	// always
	SIf.Cur.dinPosition_0_1deg := LREAL_TO_DINT(In_pAD_SIf^.stMove.lreActPos)*10;
	SIf.Cur.dinModPosition_0_1deg := LREAL_TO_DINT(In_pAD_SIf^.stMove.lreActModPos)*10;
	SIf.Cur.dinSpeed_0_1deg_s := LREAL_TO_DINT(In_pAD_SIf^.stMove.lreActVel)*10;
	SIf.Cur.dinTorque_0_1Nm := LREAL_TO_DINT(In_pAD_SIf^.stMove.lreActTorque)*10;
	SIf.Cur.bol_di1 := In_pAD_SIf^.stStatus.stDigIn.bol_SI0;
	SIf.Cur.bol_di2 := In_pAD_SIf^.stStatus.stDigIn.bol_SI1;
	SIf.Cur.bol_di3 := In_pAD_SIf^.stStatus.stDigIn.bol_SI2;
	SIf.Cur.bol_di4 := In_pAD_SIf^.stStatus.stDigIn.bol_SI3; // used for homing.....

	// info message 'software limit reached'
	IF ((In_pAD_SIf^.stStatus.bolNegSWSwitch) OR (In_pAD_SIf^.stStatus.bolPosSWSwitch)) THEN 
		IF (SIf.Alm[E_ALM_RAX.SwLimit].bol=FALSE)THEN
			// 'software limit reached';
			pfbAlarmCtrl^.setAlarm(CIf.Info.intCtrlId,E_ALM_RAX.SwLimit,0,ADR(SIf.Alm),E_AlmState.SET,CIf.Job.eMe_ActivAlmClass);
			SIf.Alm[E_ALM_RAX.SwLimit].bol:= TRUE;
		END_IF;
	ELSE
		IF (SIf.Alm[E_ALM_RAX.SwLimit].bol) THEN
			pfbAlarmCtrl^.setAlarm(CIf.Info.intCtrlId,4,0,ADR(SIf.Alm),E_AlmState.CLR,CIf.Job.eMe_ActivAlmClass);
			SIf.Alm[E_ALM_RAX.SwLimit].bol:= FALSE;
		END_IF
	END_IF
	
	//------------------------------------------------------------------------------------------------------------------------------------
	// set parameter
	// in Manual set % speed to 100% for single cmd's
	IF (CIf.Job.eMode=E_Mode.MANU) THEN
		SIf.Par.dinSpeed_per := 100;
		SIf.Par.dinAcc_per := 100;
		SIf.Par.dinDec_per := 100;
	END_IF	
	
	In_pAD_SIf^.stMove.lreSetSpeed := fSetPar(SIf.Par.dinSpeed_0_1deg_s,SIf.Par.dinSpeed_per);
	In_pAD_SIf^.stMove.lreSetAcc := fSetPar(SIf.Par.dintAccDec_0_1deg_s2,SIf.Par.dinAcc_per);
	In_pAD_SIf^.stMove.lreSetDec := fSetPar(SIf.Par.dintAccDec_0_1deg_s2,SIf.Par.dinDec_per);
	IF (SIf.Par.dinSetDecFast_0_1deg_s2>0) THEN
		In_pAD_SIf^.stMove.lreSetDecFast := DINT_TO_LREAL(SIf.Par.dinSetDecFast_0_1deg_s2)/10.0;
	ELSE
		In_pAD_SIf^.stMove.lreSetDecFast := In_pAD_SIf^.stMove.lreSetDec;
	END_IF
	In_pAD_SIf^.stCfg.bolSimulation := CIf.SwCfg.bolSimulation;
	
	// ----------------------------------------------------------------------------------
	// Conditions Always
	IF (me.StateMachine.intState>cSTA_PON) THEN	
		IF ((In_pAD_SIf^.stErr.bolErrorActive) AND (me.StateMachine.intState<>cSTA_ERROR) AND (me.StateMachine.intState<>cSTA_ERRORQuit)) THEN
			// detect drive error
			me.StateMachine.intStateNext := cSTA_ERROR;
		END_IF
	END_IF
END_IF
END_METHOD

PROPERTY PUBLIC CtrlSIf : POINTER TO T_Ctrl_SIf_RAX
GET
CtrlSIf := ADR(SIf);
END_GET
END_PROPERTY

{attribute 'object_name' := 'FB_init'}
METHOD FB_init : BOOL
VAR_INPUT
	///if TRUE, the retain variables are initialized (warm start / cold start)
	bInitRetains: BOOL;
	///if TRUE, the instance afterwards gets moved into the copy code (online change)
	bInCopyCode: BOOL;
END_VAR
VAR
	udiTaskCnt: UDINT;
END_VAR
//------------------------------------------------------------------------------------------------------------------------
// to manually change in new FUB implementation!!!
// define valid commands for this controller
FOR ii:= 0 TO (SIZEOF(CIf.Job.aCmdList)/SIZEOF(CIf.Job.aCmdList[0])-1) BY 1 DO
	IF (CIf.Job.aCmdList[ii].intCmd=cCMD_INITIALIZED) THEN
		// found first empty array element
		EXIT;
	END_IF
END_FOR
CIf.Job.aCmdList[ii].intCmd := cCMD_INIT;
CIf.Job.aCmdList[ii].strName := 'Init'; 
CIf.Job.aCmdList[ii].bolAvailable := TRUE;
ii := ii +1;
CIf.Job.aCmdList[ii].intCmd := RAX_CmdState.cCMD_POS;
CIf.Job.aCmdList[ii].strName := 'Position absolute';
CIf.Job.aCmdList[ii].bolAvailable := TRUE;
ii := ii +1;
CIf.Job.aCmdList[ii].intCmd := RAX_CmdState.cCMD_JOG_NEG;
CIf.Job.aCmdList[ii].strName := 'jogging negativ direction';
CIf.Job.aCmdList[ii].bolAvailable := TRUE;
ii := ii +1;
CIf.Job.aCmdList[ii].intCmd := RAX_CmdState.cCMD_JOG_POS;
CIf.Job.aCmdList[ii].strName := 'jogging positive direction';
CIf.Job.aCmdList[ii].bolAvailable := TRUE;
ii := ii +1;
CIf.Job.aCmdList[ii].intCmd := RAX_CmdState.cCMD_HOME;
CIf.Job.aCmdList[ii].strName := 'Home';
CIf.Job.aCmdList[ii].bolAvailable := TRUE;
ii := ii +1;
CIf.Job.aCmdList[ii].intCmd := RAX_CmdState.cCMD_REL_POS;
CIf.Job.aCmdList[ii].strName := 'Relative move';
CIf.Job.aCmdList[ii].bolAvailable := TRUE;
ii := ii +1;
CIf.Job.aCmdList[ii].intCmd := RAX_CmdState.cCMD_TURN;
CIf.Job.aCmdList[ii].strName := 'Turn';
CIf.Job.aCmdList[ii].bolAvailable := TRUE;
ii := ii +1;

// set name of class/typ
CIf.Info.strType := 'FB_RAX';
CIf.Info.strFullName := 'Rotative Axis';

// set alarm class
SIf.Alm[E_ALM_RAX.GeneralDrive].eAlmClass := E_AlmClass.OFF;
SIf.Alm[E_ALM_RAX.GeneralDrive].strText := 'general drive failure -> info number'; 
SIf.Alm[E_ALM_RAX.GeneralNc].eAlmClass := E_AlmClass.OFF;
SIf.Alm[E_ALM_RAX.GeneralNc].strText := 'general nc failure -> info number';
SIf.Alm[E_ALM_RAX.SwLimit].eAlmClass := E_AlmClass.INFO;
SIf.Alm[E_ALM_RAX.SwLimit].strText := 'software limit reached';
SIf.Alm[E_ALM_RAX.NegHwLimit].eAlmClass := E_AlmClass.OFF;
SIf.Alm[E_ALM_RAX.NegHwLimit].strText := 'neg. hardware switch detected';
SIf.Alm[E_ALM_RAX.PosHwLimit].eAlmClass := E_AlmClass.OFF;
SIf.Alm[E_ALM_RAX.PosHwLimit].strText := 'pos. hardware switch detected';
SIf.Alm[E_ALM_RAX.InterlockNegMove].eAlmClass := E_AlmClass.EOFF;
SIf.Alm[E_ALM_RAX.InterlockNegMove].strText := 'interlock neg. movement - movement stopped';
SIf.Alm[E_ALM_RAX.InterlockPosMove].eAlmClass := E_AlmClass.EOFF;
SIf.Alm[E_ALM_RAX.InterlockPosMove].strText := 'interlock pos. movement  - movement stopped';
SIf.Alm[E_ALM_RAX.GeneralMCFUB].eAlmClass := E_AlmClass.STOP;
SIf.Alm[E_ALM_RAX.GeneralMCFUB].strText := 'MC fub error -> info number';

//*******************************************************************************
// initial values
//*******************************************************************************

// software configuration
CIf.SwCfg.bolExist := TRUE;
CIf.SwCfg.bolSimulation := FALSE;

// cfg
//SIf.Cfg.eHomingMode := MC_HomingMode.MC_Direct;
SIf.Cfg.eHomingMode := MC_HomingMode.MC_DefaultHoming;
SIf.Cfg.lreShortestWayWindow_deg := 20.0; //20.0°

// parmeter
SIf.Par.dinHomeOffset_0_1deg := -900;
SIf.Par.dinPos_0_1deg := 0;
SIf.Par.dinRelDist_0_1deg := 10;
SIf.Par.dinPositionInit_0_1deg := 0;
SIf.Par.dintAccDec_0_1deg_s2 := 4000;
SIf.Par.dinAcc_per := 100;
SIf.Par.dinDec_per := 100;
SIf.Par.dinSetDecFast_0_1deg_s2 := 4000;
SIf.Par.dinSpeed_0_1deg_s := 200;
SIf.Par.dinSpeed_per := 200;
SIf.Par.dinSWLimitNeg_0_1deg := 0;
SIf.Par.dinSWLimitPos_0_1deg := 360;
END_METHOD

{attribute 'object_name' := 'getCmdState'}
METHOD PROTECTED getCmdState : STRING
VAR_INPUT
	intCmdState: INT;
	bolState: BOOL;
END_VAR
getCmdState := SUPER^.getCmdState(intCmdState:=intCmdState,bolState:=bolState); // get global/base defined cmds/states
IF (getCmdState='') THEN // global not defined get local
	// get string cmd/state string information in runtime
	IF (bolState=FALSE) THEN
		// cmd's
		CASE intCmdState OF
			RAX_CmdState.cCMD_HOME: 
				getCmdState := 'cCMD_HOME';
			RAX_CmdState.cCMD_POS: 
				getCmdState := 'cCMD_POS';
			RAX_CmdState.cCMD_JOG_NEG: 
				getCmdState := 'cCMD_JOG_NEG';
			RAX_CmdState.cCMD_JOG_POS: 
				getCmdState := 'cCMD_JOG_POS';
			RAX_CmdState.cCMD_REL_POS: 
				getCmdState := 'cCMD_REL_POS';
			RAX_CmdState.cCMD_TURN: 
				getCmdState := 'cCMD_TURN';
		ELSE
				getCmdState := 'not defined';
		END_CASE;
	ELSE
	
	// cmd's
		CASE intCmdState OF
			RAX_CmdState.cSTA_POSBusy: 
				getCmdState := 'cSTA_POSBusy';
			RAX_CmdState.cSTA_POS: 
				getCmdState := 'cSTA_POS';
			RAX_CmdState.cSTA_JOG_NEG: 
				getCmdState := 'cSTA_JOG_NEG';
			RAX_CmdState.cSTA_JOG_POS: 
				getCmdState := 'cSTA_JOG_POS';
			RAX_CmdState.cSTA_REL_POSBusy: 
				getCmdState := 'cSTA_REL_POSBusy';
			RAX_CmdState.cSTA_REL_POS: 
				getCmdState := 'cSTA_REL_POS';
			RAX_CmdState.cSTA_TURNBusy: 
				getCmdState := 'cSTA_TURNBusy';
			RAX_CmdState.cSTA_TURN: 
				getCmdState := 'cSTA_TURN';			
			cSUB_WriteSW: 
				getCmdState := 'cSUB_WriteSW';
			cSUB_Home: 
				getCmdState := 'cSUB_Home';
			cSUB_MoveToInitPos: 
				getCmdState := 'cSUB_MoveToInitPos';
			cSUB_Finished: 
				getCmdState := 'cSUB_Finished';
			cSUB_INITIALIZED:
				getCmdState := 'cSUB_INITIALIZED';
		ELSE
				getCmdState := 'not defined';
		END_CASE;
	END_IF
END_IF
END_METHOD

{attribute 'object_name' := 'getDirection'}
METHOD PROTECTED getDirection : MC_Direction
VAR_INPUT
	dinActualPosition: DINT;
	lreSetPosition: LREAL;
END_VAR
VAR
	Direction: MC_Direction;
	lreActualPosition: LREAL;
END_VAR
Direction := MC_Positive_Direction;	// MC_Shortest_Way, MC_Negative_Direction, 
lreActualPosition := DINT_TO_LREAL(dinActualPosition)/10.0;
IF (ABS(ABS(lreActualPosition) - ABS(lreSetPosition)) <= SIf.Cfg.lreShortestWayWindow_deg) THEN
	Direction := MC_Shortest_Way;
ELSIF (lreActualPosition < 0) THEN
	Direction := MC_Negative_Direction;
END_IF;

getDirection := Direction;
END_METHOD

{attribute 'object_name' := 'IoOutBridge'}
METHOD PROTECTED IoOutBridge : BOOL
// digitale and analoge inputs read from hardware or forcing
IF (CIf.SwCfg.bolSimulation = FALSE) THEN
	// check interlocks to prevent damages
	IF (CIf.Job.bolIlkOverwrite=FALSE) THEN
		IF (SIf.Ilk.bolMovePos) AND (In_pAD_SIf^.stStatus.bolCtrlOn)  AND ((In_pAD_SIf^.intCmd=cPOD_CMD_POS_JOG) OR (In_pAD_SIf^.intCmd=cPOD_CMD_POS_MOVE) OR
			((In_pAD_SIf^.stMove.lreSetPos > In_pAD_SIf^.stMove.lreActPos) AND (In_pAD_SIf^.intCmd=cPOD_CMD_ABS_MOVE)) OR
			((In_pAD_SIf^.intCmd=cPOD_CMD_REL_MOVE) AND (In_pAD_SIf^.stMove.lreSetPos>0)) OR (SIf.Cur.dinSpeed_0_1deg_s>5)  )THEN	
			// SIf.Alm[8].strText := 'interlock pos. movement  - movement stopped';
			pfbAlarmCtrl^.setAlarm(CIf.Info.intCtrlId,E_ALM_RAX.InterlockPosMove,0,ADR(SIf.Alm),E_AlmState.RST,CIf.Job.eMe_ActivAlmClass);
			In_pAD_SIf^.intCmd:=cPOD_CMD_EMCY_STOP_CTRL_OFF;
		END_IF
		IF (SIf.Ilk.bolMoveNeg) AND (In_pAD_SIf^.stStatus.bolCtrlOn)  AND ((In_pAD_SIf^.intCmd=cPOD_CMD_NEG_JOG) OR (In_pAD_SIf^.intCmd=cPOD_CMD_NEG_MOVE) OR
		 	(In_pAD_SIf^.intCmd=cPOD_CMD_HOME) OR
			((In_pAD_SIf^.stMove.lreSetPos < In_pAD_SIf^.stMove.lreActPos) AND (In_pAD_SIf^.intCmd=cPOD_CMD_ABS_MOVE)) OR
			((In_pAD_SIf^.intCmd=cPOD_CMD_REL_MOVE) AND (In_pAD_SIf^.stMove.lreSetPos<0)) OR (SIf.Cur.dinSpeed_0_1deg_s<-5)  )THEN		
			// 'interlock neg. movement - movement stopped';
			pfbAlarmCtrl^.setAlarm(CIf.Info.intCtrlId,E_ALM_RAX.InterlockNegMove,0,ADR(SIf.Alm),E_AlmState.RST,CIf.Job.eMe_ActivAlmClass);
			In_pAD_SIf^.intCmd:=cPOD_CMD_EMCY_STOP_CTRL_OFF;
		END_IF	
	END_IF

END_IF
END_METHOD

{attribute 'object_name' := 'sta_EOFF'}
METHOD PROTECTED sta_EOFF : BOOL
// state implemetation
//--------------------------------------------------------------------------------------
// Entry action
	IF (me.StateMachine.intState<>me.StateMachine.intStateLastCycle) THEN
		me.StateMachine.intStateLastCycle := me.StateMachine.intState;
		
	END_IF


//--------------------------------------------------------------------------------------
// Cyclic action
	IF (me.StateMachine.intState=me.StateMachine.intStateLastCycle) THEN
		
		// State Change Condition
		IF (me.intCmd<>cCMD_EOFF) AND (me.intCmd<>cCMD_DONE)  AND (me.Alarm.eActivAlmClass<>E_AlmClass.EOFF) THEN
			me.StateMachine.intStateNext := cSTA_OFFBusy;
		END_IF
	END_IF




//--------------------------------------------------------------------------------------
// Exit action
	IF (me.StateMachine.intState<>me.StateMachine.intStateNext) THEN
		;
	END_IF
END_METHOD

{attribute 'object_name' := 'sta_EOFFBusy'}
METHOD PROTECTED sta_EOFFBusy : BOOL
// state implemetation
//--------------------------------------------------------------------------------------
// Entry action
	IF (me.StateMachine.intState<>me.StateMachine.intStateLastCycle) THEN
		me.StateMachine.intStateLastCycle := me.StateMachine.intState;
				
		In_pAD_SIf^.intCmd := cPOD_CMD_EMCY_STOP_CTRL_OFF;
		
	END_IF


//--------------------------------------------------------------------------------------
// Cyclic action
	IF (me.StateMachine.intState=me.StateMachine.intStateLastCycle) THEN
		
		// Simulation
		IF (CIf.SwCfg.bolSimulation) THEN
			;
		END_IF
	
		// no change action
	
		// State Change Condition
		IF (In_pAD_SIf^.intCmd=cPOD_CMD_DONE) AND (In_pAD_SIf^.stStatus.bolCtrlOn=FALSE) THEN
			me.StateMachine.intStateNext := cSTA_EOFF;
		END_IF
	END_IF




//--------------------------------------------------------------------------------------
// Exit action
	IF (me.StateMachine.intState<>me.StateMachine.intStateNext) THEN
		;
	END_IF
END_METHOD

{attribute 'object_name' := 'sta_ERROR'}
METHOD PROTECTED sta_ERROR : BOOL
// state implemetation
//--------------------------------------------------------------------------------------
// Entry action
	IF (me.StateMachine.intState<>me.StateMachine.intStateLastCycle) THEN
		me.StateMachine.intStateHistory := me.StateMachine.intStateLastCycle; // -> possibillity to go back to state before error
		me.StateMachine.intStateLastCycle := me.StateMachine.intState;
		
		
		IF (In_pAD_SIf^.stErr.bolNCError) THEN
			// := 'general nc failure -> info number';
			pfbAlarmCtrl^.setAlarm(CIf.Info.intCtrlId,E_ALM_RAX.GeneralNc,DWORD_TO_DINT(In_pAD_SIf^.stErr.dwoErrorID),ADR(SIf.Alm),E_AlmState.RST,CIf.Job.eMe_ActivAlmClass);
		ELSIF (In_pAD_SIf^.stErr.bolMCError) THEN // to define
			//'MC fub error -> info number';
			pfbAlarmCtrl^.setAlarm(CIf.Info.intCtrlId,E_ALM_RAX.GeneralMCFUB,DWORD_TO_DINT(In_pAD_SIf^.stErr.dwoErrorID),ADR(SIf.Alm),E_AlmState.RST,CIf.Job.eMe_ActivAlmClass);
		ELSIF(In_pAD_SIf^.stErr.dwoErrorID=32000) THEN // Limit switch during movement
			IF (In_pAD_SIf^.stStatus.bolNegHWSwitch) THEN
				// 'neg. hardware switch detected';
				pfbAlarmCtrl^.setAlarm(CIf.Info.intCtrlId,E_ALM_RAX.NegHwLimit,0,ADR(SIf.Alm),E_AlmState.RST,CIf.Job.eMe_ActivAlmClass);
			ELSE
				// 'pos. hardware switch detected';
				pfbAlarmCtrl^.setAlarm(CIf.Info.intCtrlId,E_ALM_RAX.PosHwLimit,0,ADR(SIf.Alm),E_AlmState.RST,CIf.Job.eMe_ActivAlmClass);
			END_IF
		ELSE
			// 'general drive failure -> info number'; 
			pfbAlarmCtrl^.setAlarm(CIf.Info.intCtrlId,E_ALM_RAX.GeneralDrive,DWORD_TO_DINT(In_pAD_SIf^.stErr.dwoErrorID),ADR(SIf.Alm),E_AlmState.RST,CIf.Job.eMe_ActivAlmClass);
		END_IF
			
	END_IF


//--------------------------------------------------------------------------------------
// Cyclic action
	IF (me.StateMachine.intState=me.StateMachine.intStateLastCycle) THEN

		// State Change Condition
		IF (CIf.Job.bolAlmReset = TRUE) THEN
			me.StateMachine.intStateNext := cSTA_ERRORQuit;
		END_IF
	END_IF




//--------------------------------------------------------------------------------------
// Exit action
	IF (me.StateMachine.intState<>me.StateMachine.intStateNext) THEN
		;
	END_IF
END_METHOD

{attribute 'object_name' := 'sta_ERRORQuit'}
METHOD PROTECTED sta_ERRORQuit : BOOL
// state implemetation
//--------------------------------------------------------------------------------------
// Entry action
	IF (me.StateMachine.intState<>me.StateMachine.intStateLastCycle) THEN
		me.StateMachine.intStateLastCycle := me.StateMachine.intState;
		
	END_IF


//--------------------------------------------------------------------------------------
// Cyclic action
	IF (me.StateMachine.intState=me.StateMachine.intStateLastCycle) THEN
		
		;
		// evtl. wait time if reset of device is necessary and then decide to go to states or ERROR state
		IF (CIf.Job.bolAlmReset = TRUE) THEN
			In_pAD_SIf^.stErr.bolErrAck := TRUE; // reset drive error
			CIf.Job.eMe_ActivAlmClass := E_AlmClass.NONE; // reset feedback channel for parent
			CIf.Job.bolAlmReset := FALSE;
		END_IF
		
		// State Change Condition
		IF (In_pAD_SIf^.stErr.bolErrAck = FALSE) THEN // reset done on drive
			IF (me.StateMachine.intStateHistory<=cSTA_PON) THEN
				me.StateMachine.intStateNext := cSTA_PONBusy;
			ELSE
				me.StateMachine.intStateNext := cSTA_OFFBusy;
			END_IF
		END_IF
	END_IF




//--------------------------------------------------------------------------------------
// Exit action
	IF (me.StateMachine.intState<>me.StateMachine.intStateNext) THEN
		;
	END_IF
END_METHOD

{attribute 'object_name' := 'sta_INIT'}
METHOD PROTECTED sta_INIT : BOOL
// state implemetation
//--------------------------------------------------------------------------------------
// Entry action
	IF (me.StateMachine.intState<>me.StateMachine.intStateLastCycle) THEN
		me.StateMachine.intStateLastCycle := me.StateMachine.intState;
		
	END_IF


//--------------------------------------------------------------------------------------
// Cyclic action
	IF (me.StateMachine.intState=me.StateMachine.intStateLastCycle) THEN
		
		;
		
		// State Change Condition
		// check if no important alarm activ
		IF (me.intCmd=RAX_CmdState.cCMD_POS) THEN 
			me.StateMachine.intStateNext := RAX_CmdState.cSTA_POSBusy;
		ELSIF(me.intCmd=RAX_CmdState.cCMD_REL_POS) THEN
				me.StateMachine.intStateNext := RAX_CmdState.cSTA_REL_POSBusy;
		ELSIF(me.intCmd=RAX_CmdState.cCMD_JOG_NEG) THEN
			me.StateMachine.intStateNext := RAX_CmdState.cSTA_JOG_NEG;
		ELSIF(me.intCmd=RAX_CmdState.cCMD_JOG_POS) THEN
			me.StateMachine.intStateNext := RAX_CmdState.cSTA_JOG_POS;
		ELSIF (me.intCmd=RAX_CmdState.cCMD_TURN) THEN 
			me.StateMachine.intStateNext := RAX_CmdState.cSTA_TURNBusy;
		ELSIF (me.intCmd=cCMD_STOP) THEN 
			me.StateMachine.intStateNext := cSTA_STOPBusy;
		END_IF
	END_IF




//--------------------------------------------------------------------------------------
// Exit action
	IF (me.StateMachine.intState<>me.StateMachine.intStateNext) THEN
		;
	END_IF
END_METHOD

{attribute 'object_name' := 'sta_INITBusy'}
METHOD PROTECTED sta_INITBusy : BOOL
// state implemetation
//--------------------------------------------------------------------------------------
// Entry action
	IF (me.StateMachine.intState<>me.StateMachine.intStateLastCycle) THEN
		me.StateMachine.intStateLastCycle := me.StateMachine.intState;

		me.SubStateMachine.intState := cSUB_INITIALIZED; // reset sub statemachine
		me.SubStateMachine.intStateLastCycle := me.SubStateMachine.intState-1;
		me.SubStateMachine.intStateNext := me.SubStateMachine.intState;	
	END_IF


//--------------------------------------------------------------------------------------
// Cyclic action
	IF (me.StateMachine.intState=me.StateMachine.intStateLastCycle) THEN
		
		// Simulation
		IF (CIf.SwCfg.bolSimulation) THEN
			;
		END_IF
	
		// no change action
		// ---------------------------------------------------------------------------------------------------------------------------
		// sub state machine for sequence
		CASE me.SubStateMachine.intState OF
			//--------------------------------------------------------------------------------------
			cSUB_INITIALIZED:
				// Entry action
				IF (me.SubStateMachine.intState<>me.SubStateMachine.intStateLastCycle) THEN
					me.SubStateMachine.intStateLastCycle := me.SubStateMachine.intState;
				END_IF	
				
				// -------------------------------- State Change Condition
				IF(TRUE) THEN
					me.SubStateMachine.intStateNext := cSUB_WriteSW;
				END_IF
					
			//--------------------------------------------------------------------------------------
			cSUB_WriteSW:
				// Entry action
				IF (me.SubStateMachine.intState<>me.SubStateMachine.intStateLastCycle) THEN
					me.SubStateMachine.intStateLastCycle := me.SubStateMachine.intState;
				END_IF	
				
				(*
				// write sw offset to nc system offset to real axis system/encoder!!!!!!!!
				IF ((SIf.Par.lreHomeOffset_mm<>In_pAD_SIf^.stcfg.lreHomePosition) AND (In_pAD_SIf^.intServiceCmd=cPOD_CMD_DONE)) THEN
					In_pAD_SIf^.stService.eNC_ParNumber := MC_AxisParameter.AxisEncoderOffset;
					In_pAD_SIf^.stService.strValue := LREAL_TO_STRING(SIf.Par.lreHomeOffset_mm);
					In_pAD_SIf^.intServiceCmd := cPOD_SCMD_WRITE_PARA_NC;
					In_pAD_SIf^.stcfg.lreHomePosition := SIf.Par.lreHomeOffset_mm;
				END_IF
				
				// write sw-limits to nc system
				IF ((SIf.Par.lreSWLimitNeg_mm<>In_pAD_SIf^.stMove.lreSWLimitNeg_mm) AND (In_pAD_SIf^.intServiceCmd=cPOD_CMD_DONE)) THEN
					In_pAD_SIf^.stService.eNC_ParNumber := MC_AxisParameter.SWLimitNeg;
					In_pAD_SIf^.stService.strValue := LREAL_TO_STRING(SIf.Par.lreSWLimitNeg_mm);
					In_pAD_SIf^.intServiceCmd := cPOD_SCMD_WRITE_PARA_NC;
					In_pAD_SIf^.stMove.lreSWLimitNeg_mm := SIf.Par.lreSWLimitNeg_mm;
				END_IF
				
				IF ((SIf.Par.lreSWLimitPos_mm<>In_pAD_SIf^.stMove.lreSWLimitPos_mm) AND (In_pAD_SIf^.intServiceCmd=cPOD_CMD_DONE)) THEN
					In_pAD_SIf^.stService.eNC_ParNumber := MC_AxisParameter.SWLimitPos;
					In_pAD_SIf^.stService.strValue := LREAL_TO_STRING(SIf.Par.lreSWLimitPos_mm);
					In_pAD_SIf^.intServiceCmd := cPOD_SCMD_WRITE_PARA_NC;
					In_pAD_SIf^.stMove.lreSWLimitPos_mm := SIf.Par.lreSWLimitPos_mm;
				END_IF
*)
				// -------------------------------- State Change Condition
				IF (In_pAD_SIf^.intServiceCmd=cPOD_CMD_DONE) THEN
					IF ((me.intCmd=RAX_CmdState.cCMD_HOME) OR (In_pAD_SIf^.stStatus.bolHomeOk=FALSE)) THEN
						me.SubStateMachine.intStateNext := cSUB_Home;
					ELSIF (me.intCmd=cCMD_INIT) THEN
						me.SubStateMachine.intStateNext := cSUB_MoveToInitPos;
					ELSE
						me.SubStateMachine.intStateNext := cSUB_Finished; // no movement to init position no cmd INIT or HOME
					END_IF;
				END_IF
					
			//--------------------------------------------------------------------------------------
			cSUB_Home:
				// Entry action
				IF (me.SubStateMachine.intState<>me.SubStateMachine.intStateLastCycle) THEN
					me.SubStateMachine.intStateLastCycle := me.SubStateMachine.intState;
		
					In_pAD_SIf^.stCfg.eHomingMode := SIf.Cfg.eHomingMode;
					In_pAD_SIf^.stCfg.lreHomePosition := DINT_TO_LREAL(SIf.Par.dinHomeOffset_0_1deg)/10.0;
					In_pAD_SIf^.intCmd := cPOD_CMD_HOME;	// start homing
	
				END_IF
					
				// State Change Condition
				IF (In_pAD_SIf^.stStatus.bolHomeOk) AND (In_pAD_SIf^.intCmd=cPOD_CMD_DONE) THEN
					me.SubStateMachine.intStateNext := cSUB_MoveToInitPos;
				END_IF
				
			//--------------------------------------------------------------------------------------
			cSUB_MoveToInitPos:
				// Entry action
				IF (me.SubStateMachine.intState<>me.SubStateMachine.intStateLastCycle) THEN
					me.SubStateMachine.intStateLastCycle := me.SubStateMachine.intState;
				
					In_pAD_SIf^.stMove.lreSetPos := DINT_TO_LREAL(SIf.Par.dinPositionInit_0_1deg)/10.0;
					In_pAD_SIf^.stMove.eDirection := getDirection(dinActualPosition:=SIf.Cur.dinModPosition_0_1deg,lreSetPosition:=In_pAD_SIf^.stMove.lreSetPos);
					//In_pAD_SIf^.intCmd := cPOD_CMD_MOD_MOVE;	// absolute position
					In_pAD_SIf^.intCmd := cPOD_CMD_ABS_MOVE;	// absolute position
				END_IF
						
				// State Change Condition
				IF (In_pAD_SIf^.stStatus.bolInPos) AND (In_pAD_SIf^.intCmd=cPOD_CMD_DONE) THEN
					me.SubStateMachine.intStateNext := cSUB_Finished;
				END_IF
				
			//--------------------------------------------------------------------------------------
			cSUB_Finished:
				// Entry action
				IF (me.SubStateMachine.intState<>me.SubStateMachine.intStateLastCycle) THEN
					me.SubStateMachine.intStateLastCycle := me.SubStateMachine.intState;
				END_IF
		END_CASE
		
		// State Change Condition
		IF (me.SubStateMachine.intState =cSUB_Finished) THEN
			me.StateMachine.intStateNext := cSTA_INIT;
		END_IF
	END_IF




//--------------------------------------------------------------------------------------
// Exit action
	IF (me.StateMachine.intState<>me.StateMachine.intStateNext) THEN
		CIf.Job.strSubState := '';
	END_IF
END_METHOD

{attribute 'object_name' := 'sta_JOG_NEG'}
METHOD PROTECTED sta_JOG_NEG : BOOL
// state implemetation
//--------------------------------------------------------------------------------------
// Entry action
	IF (me.StateMachine.intState<>me.StateMachine.intStateLastCycle) THEN
		me.StateMachine.intStateLastCycle := me.StateMachine.intState;

	END_IF


//--------------------------------------------------------------------------------------
// Cyclic action
	IF (me.StateMachine.intState=me.StateMachine.intStateLastCycle) THEN

		// Simulation
		IF (CIf.SwCfg.bolSimulation) THEN
			;
		END_IF
		
		In_pAD_SIf^.intCmd := cPOD_CMD_NEG_JOG;
		
		// State Change Condition
		IF (me.intCmd=RAX_CmdState.cCMD_JOG_POS) THEN
			me.StateMachine.intStateNext := RAX_CmdState.cSTA_JOG_POS;
		ELSIF (me.intCmd<>RAX_CmdState.cCMD_JOG_NEG) AND (me.intCmd<>cCMD_DONE) THEN
			me.StateMachine.intStateNext := cSTA_STOPBusy;
		END_IF
	END_IF


//--------------------------------------------------------------------------------------
// Exit action
	IF (me.StateMachine.intState<>me.StateMachine.intStateNext) THEN
		;
	END_IF
END_METHOD

{attribute 'object_name' := 'sta_JOG_POS'}
METHOD PROTECTED sta_JOG_POS : BOOL
// state implemetation
//--------------------------------------------------------------------------------------
// Entry action
	IF (me.StateMachine.intState<>me.StateMachine.intStateLastCycle) THEN
		me.StateMachine.intStateLastCycle := me.StateMachine.intState;

	END_IF


//--------------------------------------------------------------------------------------
// Cyclic action
	IF (me.StateMachine.intState=me.StateMachine.intStateLastCycle) THEN

		// Simulation
		IF (CIf.SwCfg.bolSimulation) THEN
			;
		END_IF
		
		//no change action
		In_pAD_SIf^.intCmd := cPOD_CMD_POS_JOG;
		
		// State Change Condition
		IF (me.intCmd=RAX_CmdState.cCMD_JOG_NEG) THEN
			me.StateMachine.intStateNext := RAX_CmdState.cSTA_JOG_NEG;
		ELSIF (me.intCmd<>RAX_CmdState.cCMD_JOG_POS) AND (me.intCmd<>cCMD_DONE) THEN
			me.StateMachine.intStateNext := cSTA_STOPBusy;
		END_IF
	END_IF


//--------------------------------------------------------------------------------------
// Exit action
	IF (me.StateMachine.intState<>me.StateMachine.intStateNext) THEN
		;
	END_IF
END_METHOD

{attribute 'object_name' := 'sta_OFF'}
METHOD PROTECTED sta_OFF : BOOL
// state implemetation
//--------------------------------------------------------------------------------------
// Entry action
	IF (me.StateMachine.intState<>me.StateMachine.intStateLastCycle) THEN
		me.StateMachine.intStateLastCycle := me.StateMachine.intState;
		
	END_IF


//--------------------------------------------------------------------------------------
// Cyclic action
	IF (me.StateMachine.intState=me.StateMachine.intStateLastCycle) THEN
		
		;
		
		// State Change Condition
		// check if no important alarm activ
		IF (me.Alarm.eActivAlmClass<>E_AlmClass.OFF) THEN
			IF ((me.intCmd<>cCMD_OFF) AND (me.intCmd<>cCMD_DONE)) THEN 
				me.StateMachine.intStateNext := cSTA_INITBusy;
			END_IF
		END_IF
	END_IF




//--------------------------------------------------------------------------------------
// Exit action
	IF (me.StateMachine.intState<>me.StateMachine.intStateNext) THEN
		;
	END_IF
END_METHOD

{attribute 'object_name' := 'sta_OFFBusy'}
METHOD PROTECTED sta_OFFBusy : BOOL
// state implemetation
//--------------------------------------------------------------------------------------
// Entry action
	IF (me.StateMachine.intState<>me.StateMachine.intStateLastCycle) THEN
		me.StateMachine.intStateLastCycle := me.StateMachine.intState;
				
		In_pAD_SIf^.intCmd := cPOD_CMD_CTRL_OFF;	//1004;		// Switch controller off 
		
	END_IF


//--------------------------------------------------------------------------------------
// Cyclic action
	IF (me.StateMachine.intState=me.StateMachine.intStateLastCycle) THEN
		
		// Simulation
		IF (CIf.SwCfg.bolSimulation) THEN
			;
		END_IF
	
		// no change action
	
		// State Change Condition
		IF (In_pAD_SIf^.intCmd=cPOD_CMD_DONE) AND (In_pAD_SIf^.stStatus.bolCtrlOn=FALSE) THEN
			me.StateMachine.intStateNext := cSTA_OFF;
		END_IF
	END_IF




//--------------------------------------------------------------------------------------
// Exit action
	IF (me.StateMachine.intState<>me.StateMachine.intStateNext) THEN
		;
	END_IF
END_METHOD

{attribute 'object_name' := 'sta_POS'}
METHOD PROTECTED sta_POS : BOOL
// state implemetation
//--------------------------------------------------------------------------------------
// Entry action
	IF (me.StateMachine.intState<>me.StateMachine.intStateLastCycle) THEN
		me.StateMachine.intStateLastCycle := me.StateMachine.intState;

	END_IF


//--------------------------------------------------------------------------------------
// Cyclic action
	IF (me.StateMachine.intState=me.StateMachine.intStateLastCycle) THEN

		// Simulation
		IF (CIf.SwCfg.bolSimulation) THEN
			;
		END_IF
		
		// State Change Condition
		IF (me.Alarm.eActivAlmClass=E_AlmClass.STOP) OR	((me.intCmd<>RAX_CmdState.cCMD_POS) AND (me.intCmd<>cCMD_DONE)) THEN 
			me.StateMachine.intStateNext := cSTA_STOPBusy;
		END_IF
	END_IF




//--------------------------------------------------------------------------------------
// Exit action
	IF (me.StateMachine.intState<>me.StateMachine.intStateNext) THEN
		;
	END_IF
END_METHOD

{attribute 'object_name' := 'sta_POSBusy'}
METHOD PROTECTED sta_POSBusy : BOOL
// state implemetation
//--------------------------------------------------------------------------------------
// Entry action
	IF (me.StateMachine.intState<>me.StateMachine.intStateLastCycle) THEN
		me.StateMachine.intStateLastCycle := me.StateMachine.intState;
		
		In_pAD_SIf^.stMove.lreSetPos := DINT_TO_LREAL(SIf.Par.dinPos_0_1Deg)/10.0;
		In_pAD_SIf^.intCmd := cPOD_CMD_ABS_MOVE;	// start move with absolute target position 
	END_IF


//--------------------------------------------------------------------------------------
// Cyclic action
	IF (me.StateMachine.intState=me.StateMachine.intStateLastCycle) THEN

		// Simulation
		IF (CIf.SwCfg.bolSimulation) THEN
			;
		END_IF
		
		
		// State Change Condition
		IF (In_pAD_SIf^.intCmd=cPOD_CMD_DONE) AND (In_pAD_SIf^.stStatus.bolInPos) THEN
			me.StateMachine.intStateNext := RAX_CmdState.cSTA_POS;
		ELSIF (me.Alarm.eActivAlmClass=E_AlmClass.STOP) OR ((me.intCmd<>RAX_CmdState.cCMD_POS) AND (me.intCmd<>cCMD_DONE)) THEN 
			me.StateMachine.intStateNext := cSTA_STOPBusy;
		END_IF
	END_IF




//--------------------------------------------------------------------------------------
// Exit action
	IF (me.StateMachine.intState<>me.StateMachine.intStateNext) THEN
		;
	END_IF
END_METHOD

{attribute 'object_name' := 'sta_REL_POS'}
METHOD PROTECTED sta_REL_POS : BOOL
// state implemetation
//--------------------------------------------------------------------------------------
// Entry action
	IF (me.StateMachine.intState<>me.StateMachine.intStateLastCycle) THEN
		me.StateMachine.intStateLastCycle := me.StateMachine.intState;

	END_IF


//--------------------------------------------------------------------------------------
// Cyclic action
	IF (me.StateMachine.intState=me.StateMachine.intStateLastCycle) THEN

		// Simulation
		IF (CIf.SwCfg.bolSimulation) THEN
			;
		END_IF
		
		// State Change Condition
		IF (me.Alarm.eActivAlmClass=E_AlmClass.STOP) OR	((me.intCmd<>RAX_CmdState.cCMD_REL_POS) AND (me.intCmd<>cCMD_DONE)) THEN 
			me.StateMachine.intStateNext := cSTA_STOPBusy;
		END_IF
	END_IF




//--------------------------------------------------------------------------------------
// Exit action
	IF (me.StateMachine.intState<>me.StateMachine.intStateNext) THEN
		;
	END_IF
END_METHOD

{attribute 'object_name' := 'sta_REL_POSBusy'}
METHOD PROTECTED sta_REL_POSBusy : BOOL
// state implemetation
//--------------------------------------------------------------------------------------
// Entry action
	IF (me.StateMachine.intState<>me.StateMachine.intStateLastCycle) THEN
		me.StateMachine.intStateLastCycle := me.StateMachine.intState;
		
		In_pAD_SIf^.stMove.lreSetPos := DINT_TO_LREAL(SIf.Par.dinRelDist_0_1deg)/10.0; // for rel movement used also SetPos
		In_pAD_SIf^.intCmd := cPOD_CMD_REL_MOVE;	// start move with absolute target position 
	END_IF


//--------------------------------------------------------------------------------------
// Cyclic action
	IF (me.StateMachine.intState=me.StateMachine.intStateLastCycle) THEN

		// Simulation
		IF (CIf.SwCfg.bolSimulation) THEN
			;
		END_IF
		
		
		// State Change Condition
		IF (In_pAD_SIf^.intCmd=cPOD_CMD_DONE) AND (In_pAD_SIf^.stStatus.bolInPos) THEN
			me.StateMachine.intStateNext := RAX_CmdState.cSTA_REL_POS;
		ELSIF (me.Alarm.eActivAlmClass=E_AlmClass.STOP) OR ((me.intCmd<>RAX_CmdState.cCMD_REL_POS) AND (me.intCmd<>cCMD_DONE)) THEN 
			me.StateMachine.intStateNext := cSTA_STOPBusy;
		END_IF
	END_IF




//--------------------------------------------------------------------------------------
// Exit action
	IF (me.StateMachine.intState<>me.StateMachine.intStateNext) THEN
		;
	END_IF
END_METHOD

{attribute 'object_name' := 'sta_STOP'}
METHOD PROTECTED sta_STOP : BOOL
// state implemetation
//--------------------------------------------------------------------------------------
// Entry action
	IF (me.StateMachine.intState<>me.StateMachine.intStateLastCycle) THEN
		me.StateMachine.intStateLastCycle := me.StateMachine.intState;
		
	END_IF


//--------------------------------------------------------------------------------------
// Cyclic action
	IF (me.StateMachine.intState=me.StateMachine.intStateLastCycle) THEN
		
		;
		
		
		// State Change Condition
		IF (me.Alarm.eActivAlmClass<>E_AlmClass.STOP) THEN
			IF ((me.intCmd=RAX_CmdState.cCMD_HOME) OR (me.intCmd=cCMD_INIT)) THEN
				me.StateMachine.intStateNext := cSTA_INITBusy;
			ELSIF (me.intCmd=RAX_CmdState.cCMD_POS) THEN 
				me.StateMachine.intStateNext := RAX_CmdState.cSTA_POSBusy;
			ELSIF(me.intCmd=RAX_CmdState.cCMD_REL_POS) THEN
				me.StateMachine.intStateNext := RAX_CmdState.cSTA_REL_POSBusy;
			ELSIF(me.intCmd=RAX_CmdState.cCMD_JOG_NEG) THEN
				me.StateMachine.intStateNext := RAX_CmdState.cSTA_JOG_NEG;
			ELSIF(me.intCmd=RAX_CmdState.cCMD_JOG_POS) THEN
				me.StateMachine.intStateNext := RAX_CmdState.cSTA_JOG_POS;
			ELSIF(me.intCmd=RAX_CmdState.cCMD_TURN) THEN
				me.StateMachine.intStateNext := RAX_CmdState.cSTA_TURNBusy;
			END_IF
		END_IF
	END_IF




//--------------------------------------------------------------------------------------
// Exit action
	IF (me.StateMachine.intState<>me.StateMachine.intStateNext) THEN
		;
	END_IF
END_METHOD

{attribute 'object_name' := 'sta_STOPBusy'}
METHOD PROTECTED sta_STOPBusy : BOOL
// state implemetation
//--------------------------------------------------------------------------------------
// Entry action
	IF (me.StateMachine.intState<>me.StateMachine.intStateLastCycle) THEN
		me.StateMachine.intStateLastCycle := me.StateMachine.intState;
		
		In_pAD_SIf^.intCmd := cPOD_CMD_STOP;
	END_IF


//--------------------------------------------------------------------------------------
// Cyclic action
	IF (me.StateMachine.intState=me.StateMachine.intStateLastCycle) THEN
		
		
		
		// State Change Condition
		IF (In_pAD_SIf^.intCmd=cPOD_CMD_DONE) THEN
			me.StateMachine.intStateNext := cSTA_STOP;
		END_IF
	END_IF




//--------------------------------------------------------------------------------------
// Exit action
	IF (me.StateMachine.intState<>me.StateMachine.intStateNext) THEN
		;
	END_IF
END_METHOD

{attribute 'object_name' := 'sta_Turn'}
METHOD PROTECTED sta_Turn : BOOL
// state implemetation
//--------------------------------------------------------------------------------------
// Entry action
	IF (me.StateMachine.intState<>me.StateMachine.intStateLastCycle) THEN
		me.StateMachine.intStateLastCycle := me.StateMachine.intState;

	END_IF


//--------------------------------------------------------------------------------------
// Cyclic action
	IF (me.StateMachine.intState=me.StateMachine.intStateLastCycle) THEN

		// Simulation
		IF (CIf.SwCfg.bolSimulation) THEN
			;
		END_IF
		
		// State Change Condition
		IF (me.Alarm.eActivAlmClass=E_AlmClass.STOP) OR	((me.intCmd<>RAX_CmdState.cCMD_POS) AND (me.intCmd<>cCMD_DONE)) THEN 
			me.StateMachine.intStateNext := cSTA_STOPBusy;
		END_IF
	END_IF




//--------------------------------------------------------------------------------------
// Exit action
	IF (me.StateMachine.intState<>me.StateMachine.intStateNext) THEN
		;
	END_IF
END_METHOD

{attribute 'object_name' := 'sta_TurnBusy'}
METHOD PROTECTED sta_TurnBusy : BOOL
// state implemetation
//--------------------------------------------------------------------------------------
// Entry action
	IF (me.StateMachine.intState<>me.StateMachine.intStateLastCycle) THEN
		me.StateMachine.intStateLastCycle := me.StateMachine.intState;
		
		In_pAD_SIf^.stMove.lreSetPos := ABS(DINT_TO_LREAL(SIf.Par.dinPos_0_1deg)/10.0); // sign only for direction!!!!
		In_pAD_SIf^.stMove.eDirection := getDirection(dinActualPosition:=SIf.Cur.dinModPosition_0_1deg,lreSetPosition:=In_pAD_SIf^.stMove.lreSetPos);
//		In_pAD_SIf^.intCmd := cPOD_CMD_MOD_MOVE;	// start move with absolute target position 
		In_pAD_SIf^.intCmd := cPOD_CMD_ABS_MOVE;	// start move with absolute target position 
	END_IF


//--------------------------------------------------------------------------------------
// Cyclic action
	IF (me.StateMachine.intState=me.StateMachine.intStateLastCycle) THEN

		// Simulation
		IF (CIf.SwCfg.bolSimulation) THEN
			;
		END_IF
	
		// State Change Condition
		IF (In_pAD_SIf^.intCmd=cPOD_CMD_DONE) AND (In_pAD_SIf^.stStatus.bolInPos) THEN
			me.StateMachine.intStateNext := RAX_CmdState.cSTA_TURN;
		ELSIF (me.Alarm.eActivAlmClass=E_AlmClass.STOP) OR ((me.intCmd<>RAX_CmdState.cCMD_TURN) AND (me.intCmd<>cCMD_DONE)) THEN 
			me.StateMachine.intStateNext := cSTA_STOPBusy;
		END_IF
	END_IF




//--------------------------------------------------------------------------------------
// Exit action
	IF (me.StateMachine.intState<>me.StateMachine.intStateNext) THEN
		;
	END_IF
END_METHOD

{attribute 'object_name' := 'StateMachine'}
METHOD PROTECTED StateMachine : BOOL
SUPER^.StateMachine();

// main statemachine of base controller
CASE me.StateMachine.intState OF
	cSTA_INITBusy: 
        THIS^.sta_INITBusy();
    cSTA_INIT: 
        THIS^.sta_INIT();
    RAX_CmdState.cSTA_JOG_NEG: 
        THIS^.sta_JOG_NEG();
    RAX_CmdState.cSTA_JOG_POS: 
        THIS^.sta_JOG_POS();
    RAX_CmdState.cSTA_POSBusy: 
        THIS^.sta_POSBusy();
    RAX_CmdState.cSTA_POS: 
        THIS^.sta_POS();
	RAX_CmdState.cSTA_REL_POSBusy: 
        THIS^.sta_REL_POSBusy();
    RAX_CmdState.cSTA_REL_POS: 
        THIS^.sta_REL_POS();
    RAX_CmdState.cSTA_TURNBusy: 
        THIS^.sta_TurnBusy();
    RAX_CmdState.cSTA_TURN: 
        THIS^.sta_Turn();
	cSTA_STOPBusy: 
        THIS^.sta_STOPBusy();
    cSTA_STOP: 
        THIS^.sta_STOP();
END_CASE;
END_METHOD

END_FUNCTION_BLOCK

// POUs/Controller/Lvl0/RAX(Rotative Axis)/fSetPar
FUNCTION fSetPar : LREAL
VAR_INPUT
	///factor * SetValue
	In_dinSetValue: DINT;
	/// % from SetValue
	In_dinSetValue_per: DINT;
END_VAR
VAR
	/// every value is scaled with 10
	dinFactor: DINT := 10;
END_VAR

fSetPar := DINT_TO_LREAL((In_dinSetValue*In_dinSetValue_per) /(10*100));

END_FUNCTION

// POUs/Controller/Lvl1/BCH (Barcode with DataChannel)/helper/cycle_Bch
FUNCTION cycle_Bch : BOOL
VAR_INPUT
	pBch: POINTER TO T_BCH;
END_VAR

pBch^.ctrl.fbBch.In_bolSensorTrigScan := pBch^.io.In_bolSensorTrigScan;
pBch^.ctrl.fbBch();
pBch^.ctrl.fbBch_Bcc();
pBch^.ctrl.fbBch_Bcc_Bcd();
pBch^.datachn.rSendData.fbFifo();

END_FUNCTION

// POUs/Controller/Lvl1/BCH (Barcode with DataChannel)/helper/init_Bch
FUNCTION init_Bch : BOOL
VAR_INPUT
	pBch: POINTER TO T_BCH;
	/// instance array of all controller instances
	pCtrlInst: POINTER TO fb_CtrlBase;
	/// common interface array of all controllers (main use for PLC)
	pCtrlCIf: POINTER TO T_Ctrl_CIf;
END_VAR

pBch^.datachn.rSendData.fbDataChannel.InitChannel(SIZEOF(pBch^.datachn.rSendData.rDataChannelItem), ADR(pBch^.datachn.rSendData.rDataChannelItem));
pBch^.datachn.rSendData.fbFifo.DataChannel := ADR(pBch^.datachn.rSendData.fbDataChannel);
pBch^.datachn.rSendData.fbFifo.FreeDataPointer := TRUE;
pBch^.datachn.rSendData.fbFifo.Enable := TRUE;

pBch^.ctrl.fbBch_Bcc.iniAllCtrlArrays(pCtrlInst,pCtrlCIf,pBch^.id.Bch_Bcc); // init and entry fb_instance in global fb pointer array
pBch^.ctrl.fbBch_Bcc.pBCD_SIf_In := pBch^.ctrl.fbBch_Bcc_Bcd.getSIf();
pBch^.ctrl.fbBch.iniAllCtrlArrays(pCtrlInst,pCtrlCIf,pBch^.id.Bch); // init and entry fb_instance in global fb pointer array
pBch^.ctrl.fbBch.BarcodeReader := ADR(pBch^.ctrl.fbBch_Bcc);
pBch^.ctrl.fbBch.DataChannel := ADR(pBch^.datachn.rSendData.fbFifo);

END_FUNCTION

// POUs/Controller/Lvl1/BCH (Barcode with DataChannel)/FB_BCH
FUNCTION_BLOCK FB_BCH EXTENDS FB_CtrlBase
VAR_INPUT
	In_bolSensorTrigScan: BOOL;
END_VAR
VAR_OUTPUT
	Out_Barcode: ULINT;
	Out_ChangeEvent: UINT;
END_VAR
VAR
	/// Specific interface struct for public access
	SIf: T_Ctrl_SIf_BCH;
	/// Barcode Reader Variable
	p_fbBcc: POINTER TO FB_BCC;
	pBccCIf: POINTER TO T_Ctrl_CIf;
	pBccSIf: POINTER TO T_Ctrl_SIf_BCC;
	/// DataChannel
	m_pDataChannel: POINTER TO FB_DataChannelSenderFifo;
END_VAR

(*__________________________________________________________________________________________________
¦	
¦	Vistaprint Schweiz GmbH
¦	CH - 8401 Winterthur
¦
¦	www.vistaprint.ch - info@vistaprint.ch
¦___________________________________________________________________________________________________

Function desription:
ToDo: DSC...

History:
Version		Date			Author				Comment
---------------------------------------------------------------------------------------------------
0.00.1		20.05.2014		AVME/DSC			Start history. Insert all basic functionalities.
___________________________________________________________________________________________________*)


SUPER^();

{attribute 'object_name' := 'Always'}
METHOD PROTECTED Always : BOOL
// not inherite from base !!!  special behaviour for this controller
// SUPER^.Always();

// Conditions Always
IF (me.bolChangeBackToAUTO=TRUE) THEN // switch mode to automatic switch off controller
	//me.StateMachine.intStateNext := cSTA_OFFBusy;
	me.bolChangeBackToAUTO := FALSE;
END_IF

IF (CIf.SwCfg.bolExist=FALSE) THEN // hardware of controller does not exist
	me.StateMachine.intStateNext := cSTA_SINGLE_ANSWER;
ELSE
	// Handle command PON
	IF (me.intCmd=cCMD_PON) 
		AND (me.StateMachine.intState<>cSTA_PONBusy) AND (me.StateMachine.intState<>cSTA_PON)
		AND (me.StateMachine.intState<>cSTA_ERROR) AND (me.StateMachine.intState<>cSTA_ERRORQuit) 
		AND (me.StateMachine.intState<>cSTA_EOFF) AND (me.StateMachine.intState<>cSTA_EOFFBusy) THEN
		me.StateMachine.intStateNext := cSTA_PONBusy;
	END_IF
END_IF
		
// ----------------------------------------------------------------------------------
// cyclic actions outside of statemachine
IF (me.StateMachine.intState<>cSTA_SINGLE_ANSWER) THEN
	;
END_IF

// ----------------------------------------------------------------------------------
// Always change actions in Base Library
// ----------------------------------------------------------------------------------
// overrule error always from base -> no EOFF State!! in EOFF go to OFF
IF (me.StateMachine.intStateNext = cSTA_EOFFBusy) THEN
	IF (me.StateMachine.intState=cSTA_OFF) THEN
		me.StateMachine.intStateNext := cSTA_OFF;
	ELSE // stay in OFF
		me.StateMachine.intStateNext := cSTA_OFFBusy;
	END_IF
END_IF

// Conditions Always
IF (((me.Alarm.eActivAlmClass=E_AlmClass.EOFF) OR (me.Alarm.eActivAlmClass=E_AlmClass.OFF) OR (me.intCmd=cCMD_OFF))
		 AND (me.StateMachine.intState<>cSTA_ERROR) AND (me.StateMachine.intState<>cSTA_ERRORQuit) AND
		(me.StateMachine.intState<>cSTA_OFF) AND (me.StateMachine.intState<>cSTA_OFFBusy)) THEN
	// alarm evt EOFF, OFF or cmd off
	me.StateMachine.intStateNext := cSTA_OFFBusy;
END_IF
END_METHOD

PROPERTY BarcodeReader : POINTER TO FB_BCC
GET
BarcodeReader := p_fbBcc;
END_GET
SET
p_fbBcc := BarcodeReader;
END_SET
END_PROPERTY

{attribute 'object_name' := 'CtrlInit'}
METHOD CtrlInit : BOOL
SUPER^.CtrlInit();

pBccCIf := AddChild(p_fbBcc^);
pBccSIf := p_fbBcc^.getCtrlSIf();
END_METHOD

PROPERTY CtrlSIf : POINTER TO T_Ctrl_SIf_BCH
GET
CtrlSIf := ADR(SIf);
END_GET
END_PROPERTY

PROPERTY DataChannel : POINTER TO FB_DataChannelSenderFifo
SET
m_pDataChannel := DataChannel;
END_SET
END_PROPERTY

{attribute 'object_name' := 'FB_init'}
METHOD FB_init : BOOL
VAR_INPUT
	/// if TRUE, the retain variables are initialized (warm start / cold start)
	bInitRetains: BOOL;
	/// if TRUE, the instance afterwards gets moved into the copy code (online change)
	bInCopyCode: BOOL;
END_VAR
VAR
	iIdx: UINT;
	iLength: UINT;
END_VAR
// ------------------------------------------------------------------------------------------------------------------------
// to manually change in new FUB implementation!!!
// define valid commands for this controller
iLength := SIZEOF(CIf.Job.aCmdList)/SIZEOF(CIf.Job.aCmdList[0]);
iIdx := 0;

WHILE (iIdx < iLength) AND (CIf.Job.aCmdList[iIdx].intCmd <> cCMD_INITIALIZED) DO
	iIdx := iIdx + 1; 
END_WHILE

IF (iIdx < iLength) THEN
// Add configuration of own comands	
	CIf.Job.aCmdList[iIdx].intCmd := BASE_PLC.cCMD_RUN;
	CIf.Job.aCmdList[iIdx].strName := 'RUN'; 
	CIf.Job.aCmdList[iIdx].bolAvailable := TRUE;
    iIdx := iIdx + 1;
	CIf.Job.aCmdList[iIdx].intCmd := BCH_CmdState.cCMD_READ;
	CIf.Job.aCmdList[iIdx].strName := 'READ'; 
	CIf.Job.aCmdList[iIdx].bolAvailable := TRUE;
    iIdx := iIdx + 1;
ELSE
	// Error if the aCmdList Array is to small
END_IF

// set name of class/typ
CIf.Info.strType := 'FB_BCH';
CIf.Info.strFullName := 'Barcode with DataChannel';

// set alarm class
SIf.Alm[E_ALM_BCH.DataChannelMissing].eAlmClass := E_AlmClass.TSTOP;
SIf.Alm[E_ALM_BCH.DataChannelMissing].strText := 'DataChannel is missing';
SIf.Alm[E_ALM_BCH.DataChannelBufferFull].eAlmClass := E_AlmClass.TSTOP;
SIf.Alm[E_ALM_BCH.DataChannelBufferFull].strText := 'DataChannel Buffer is full';
SIf.Alm[E_ALM_BCH.BarcodeNotReadCorrectly].eAlmClass := E_AlmClass.WARNING;
SIf.Alm[E_ALM_BCH.BarcodeNotReadCorrectly].strText := 'Barcode not detected';

// *******************************************************************************
// initial values
// *******************************************************************************

// software configuration
CIf.SwCfg.bolExist := FALSE;
CIf.SwCfg.bolEnable := TRUE;
CIf.SwCfg.bolSimulation :=  FALSE;

SIf.Cfg.bolEnableDataChannel := FALSE;
SIf.Cfg.bolNegativeTriggerSignal := FALSE;
END_METHOD

{attribute 'object_name' := 'getCmdState'}
METHOD PROTECTED getCmdState : STRING
VAR_INPUT
	intCmdState: INT;
	bolState: BOOL;
END_VAR
getCmdState := SUPER^.getCmdState(intCmdState:=intCmdState,bolState:=bolState); // get global/base defined cmds/states

IF (getCmdState='') THEN // global not defined get local
	// get string cmd/state string information in runtime
	IF (bolState=FALSE) THEN
		CASE intCmdState OF
			BCH_CmdState.cCMD_READ: 
				getCmdState := 'READ';
		END_CASE;
	END_IF
END_IF
END_METHOD

{attribute 'object_name' := 'getCtrlSIf'}
METHOD getCtrlSIf : POINTER TO T_Ctrl_SIf_BCH
getCtrlSIf := ADR(SIf);
END_METHOD

{attribute 'object_name' := 'IoInBridge'}
METHOD PROTECTED IoInBridge : BOOL
// digitale and analoge inputs read from hardware or forcing
IF SIf.Cfg.bolNegativeTriggerSignal THEN
	SIf.In.bolSensorTrigScan.map			:= NOT THIS^.In_bolSensorTrigScan				;
ELSE
	SIf.In.bolSensorTrigScan.map			:= THIS^.In_bolSensorTrigScan				;
END_IF

IF (CIf.SwCfg.bolSimulation = FALSE) THEN
	BASE_PLC.getInBol(CIf.Job.bolIoForce,ADR(SIf.In.bolSensorTrigScan));
ELSE
;	//simulation of global IO
END_IF
END_METHOD

{attribute 'object_name' := 'sta_ERROR'}
METHOD PROTECTED sta_ERROR : BOOL
// state implemetation
//--------------------------------------------------------------------------------------
// Entry action
	IF (me.StateMachine.intState<>me.StateMachine.intStateLastCycle) THEN
		me.StateMachine.intStateHistory := me.StateMachine.intStateLastCycle; // -> possibillity to go back to state before error
		me.StateMachine.intStateLastCycle := me.StateMachine.intState;
	END_IF


//--------------------------------------------------------------------------------------
// Cyclic action

	// State Change Condition
	IF (CIf.Job.bolAlmReset = TRUE) THEN
		me.StateMachine.intStateNext := cSTA_ERRORQuit;
	END_IF

	
//--------------------------------------------------------------------------------------
// Exit action
	IF (me.StateMachine.intState<>me.StateMachine.intStateNext) THEN
		;
	END_IF
END_METHOD

{attribute 'object_name' := 'sta_ERRORQuit'}
METHOD PROTECTED sta_ERRORQuit : BOOL
// state implemetation
//--------------------------------------------------------------------------------------
// Entry action
	IF (me.StateMachine.intState<>me.StateMachine.intStateLastCycle) THEN
		me.StateMachine.intStateLastCycle := me.StateMachine.intState;
	END_IF


//--------------------------------------------------------------------------------------
// Cyclic action
	
	// evtl. wait time if reset of device is necessary and then decide to go to states or ERROR state
	IF (CIf.Job.bolAlmReset = TRUE) THEN
		CIf.Job.eMe_ActivAlmClass := E_AlmClass.NONE; // reset feedback channel for parent
		CIf.Job.bolAlmReset := FALSE;
		
		IF (me.StateMachine.intStateHistory=cSTA_RUN) OR (me.StateMachine.intStateHistory=cSTA_RUNBusy) THEN
			me.StateMachine.intStateNext := cSTA_RUNBusy;
		ELSE
			me.StateMachine.intStateNext := cSTA_OFFBusy;
		END_IF
		
	END_IF

	
//--------------------------------------------------------------------------------------
// Exit action
	IF (me.StateMachine.intState<>me.StateMachine.intStateNext) THEN
		;
	END_IF
END_METHOD

{attribute 'object_name' := 'sta_OFF'}
METHOD PROTECTED sta_OFF : BOOL
// state implemetation
// --------------------------------------------------------------------------------------
// Entry action
	IF (me.StateMachine.intState<>me.StateMachine.intStateLastCycle) THEN
		me.StateMachine.intStateLastCycle := me.StateMachine.intState;	
	END_IF


// --------------------------------------------------------------------------------------
// Cyclic action

	IF me.intCmd=Base_PLC.cCMD_RUN THEN
		me.StateMachine.intStateNext := Base_PLC.cSTA_RUNBusy;
	END_IF


// --------------------------------------------------------------------------------------
// Exit action
	IF (me.StateMachine.intState<>me.StateMachine.intStateNext) THEN
		;
	END_IF
END_METHOD

{attribute 'object_name' := 'sta_OFFBusy'}
METHOD PROTECTED sta_OFFBusy : BOOL
// state implemetation
// --------------------------------------------------------------------------------------
// Entry action
	IF (me.StateMachine.intState<>me.StateMachine.intStateLastCycle) THEN
		me.StateMachine.intStateLastCycle := me.StateMachine.intState;
		
		pBccCIf^.Job.intACmd := BASE_PLC.cCMD_OFF;
	END_IF


// --------------------------------------------------------------------------------------
// Cyclic action

	IF (pBccCIf^.Job.intState = BASE_PLC.cSTA_OFF) THEN
		me.StateMachine.intStateNext := cSTA_OFF;
	END_IF

	
// --------------------------------------------------------------------------------------
// Exit action
	IF (me.StateMachine.intState<>me.StateMachine.intStateNext) THEN
		;
	END_IF
END_METHOD

{attribute 'object_name' := 'sta_RUN'}
METHOD PROTECTED sta_RUN : BOOL
VAR
	uliBarcode: ULINT;
	pItem: POINTER TO T_IdBase_DCH;
END_VAR
// state implemetation
// --------------------------------------------------------------------------------------
// Entry action
	IF (me.StateMachine.intState<>me.StateMachine.intStateLastCycle) THEN
		me.StateMachine.intStateLastCycle := me.StateMachine.intState;	

		me.SubStateMachine.intState		:= BCH_CmdState.cSUB_WAITPAPER;
		me.SubStateMachine.intStateNext := BCH_CmdState.cSUB_WAITPAPER;
	END_IF


// --------------------------------------------------------------------------------------
// Cyclic action

	CASE me.SubStateMachine.intState OF
		// Wait for the paper
		// ------------------------------------------------------------------------
		BCH_CmdState.cSUB_WAITPAPER:
			IF SIf.In.bolSensorTrigScan.intern OR (me.intCmd = BCH_CmdState.cCMD_READ) THEN
				IF (me.intCmd = BCH_CmdState.cCMD_READ) THEN
					CIf.Job.intACmd := cCMD_DONE;			
					CIf.Job.intMCmd := cCMD_DONE;			
				END_IF

				me.SubStateMachine.intStateNext := BCH_CmdState.cSUB_BARCODEREADstart;
			END_IF

		// substate Start Reading Barcode
		// ------------------------------------------------------------------------
		BCH_CmdState.cSUB_BARCODEREADstart:
			pBccCIf^.Job.intACmd := BCC_CmdState.cBCC_CMD_READ;
	
			CASE pBccCIf^.Job.intState OF
				BCC_CmdState.cBCC_STA_READBusy:
					me.SubStateMachine.intStateNext := BCH_CmdState.cSUB_BARCODREREADbusy;
				cSTA_ERROR:
					me.StateMachine.intStateNext := cSTA_ERROR;
			END_CASE
	
		// substate Busy Reading Barcode
		// ------------------------------------------------------------------------
		BCH_CmdState.cSUB_BARCODREREADbusy:
			CASE pBccCIf^.Job.intState OF
				BCC_CmdState.cBCC_STA_READ:
					me.SubStateMachine.intStateNext := BCH_CmdState.cSUB_BARCODREREAD;
				cSTA_ERROR:
					me.StateMachine.intStateNext := cSTA_ERROR;
			END_CASE
	
		// substate Reading Barcode Done
		// ------------------------------------------------------------------------
		BCH_CmdState.cSUB_BARCODREREAD:
			IF SIf.Cfg.bolEnableDataChannel THEN
				IF pBccSIf^.Cur.stData.uliBarCode > 0 THEN
					uliBarcode := pBccSIf^.Cur.stData.uliBarCode;
					Out_Barcode := uliBarcode;
					Out_ChangeEvent := Out_ChangeEvent + 1;

					IF (m_pDataChannel <> NULL) AND (SIf.Cfg.bolEnableDataChannel) THEN
						IF m_pDataChannel^.ItemCount >= m_pDataChannel^.MaxFifoSize THEN
							pfbAlarmCtrl^.setAlarm(CIf.Info.intCtrlId,E_ALM_BCH.DataChannelBufferFull,0,ADR(SIf.Alm),E_AlmState.RST,CIf.Job.eMe_ActivAlmClass);
						ELSE
							pItem := __NEW(T_IdBase_DCH);
							pItem^.rBaseInfo.eHealth := E_ItemHealth.Healthy;
							pItem^.rBaseInfo.uinModuleId := 1;
							pItem^.rBaseInfo.uinActualPosition := 1;
							pItem^.udiIdentification := pBccSIf^.Cur.stData.uliBarCode;
							m_pDataChannel^.Push(pItem);					
						END_IF
					END_IF
				END_IF

				me.SubStateMachine.intStateNext := BCH_CmdState.cSUB_WAITPAPERGONE;
			END_IF
			
		// Wait Until the Paper is gone
		// ------------------------------------------------------------------------
		BCH_CmdState.cSUB_WAITPAPERGONE:
			IF NOT SIf.In.bolSensorTrigScan.intern THEN
				me.SubStateMachine.intStateNext := BCH_CmdState.cSUB_WAITPAPERGONEDELAY;
			END_IF

		// Wait Until the Paper is gone
		// ------------------------------------------------------------------------
		BCH_CmdState.cSUB_WAITPAPERGONEDELAY:
			IF me.SubStateMachine.udiTimeInState_ms > 500 THEN
				me.SubStateMachine.intStateNext := BCH_CmdState.cSUB_WAITPAPER;
			END_IF
	END_CASE

	IF me.intCmd=Base_PLC.cCMD_OFF THEN
		me.StateMachine.intStateNext := Base_PLC.cSTA_OFFBusy;
	END_IF


// --------------------------------------------------------------------------------------
// Exit action
	IF (me.StateMachine.intState<>me.StateMachine.intStateNext) THEN
		;
	END_IF
END_METHOD

{attribute 'object_name' := 'sta_RUNBusy'}
METHOD PROTECTED sta_RUNBusy : BOOL
// state implemetation
// --------------------------------------------------------------------------------------
// Entry action
	IF (me.StateMachine.intState<>me.StateMachine.intStateLastCycle) THEN
		me.StateMachine.intStateLastCycle := me.StateMachine.intState;	
	END_IF


// --------------------------------------------------------------------------------------
// Cyclic action

	IF me.intCmd=Base_PLC.cCMD_OFF THEN
		me.StateMachine.intStateNext := Base_PLC.cSTA_OFFBusy;
	ELSE
		me.StateMachine.intStateNext := Base_PLC.cSTA_RUN;
	END_IF


// --------------------------------------------------------------------------------------
// Exit action
	IF (me.StateMachine.intState<>me.StateMachine.intStateNext) THEN
		;
	END_IF
END_METHOD

{attribute 'object_name' := 'StateMachine'}
METHOD PROTECTED StateMachine : BOOL
SUPER^.StateMachine();

// main statemachine of base controller
CASE me.StateMachine.intState OF
	cSTA_RUNBusy: 
        THIS^.sta_RUNBusy();
	cSTA_RUN: 
        THIS^.sta_RUN();
END_CASE
END_METHOD

END_FUNCTION_BLOCK

// POUs/Controller/Lvl1/MDC [Malteser Drive Controller]/FB_MDC
FUNCTION_BLOCK FB_MDC EXTENDS FB_CtrlBase
VAR_INPUT
	In_bolCrossPositionSensor			: BOOL;
	In_bolTablePositionSensor			: BOOL;
END_VAR
VAR_OUTPUT
	/// Position Output to the higher controller
	Out_intActualPosition				: INT;
END_VAR
VAR
	/// Specific interface struct for public access
	SIf					: T_Ctrl_SIf_MDC;
	///pointer to function block
	p_fbMotor			: POINTER TO FB_UMC;
	pMotor_CIF			: POINTER TO BASE_PLC.T_Ctrl_CIf;
END_VAR

(*__________________________________________________________________________________________________
¦	
¦	Vistaprint Schweiz GmbH
¦	CH - 8401 Winterthur
¦
¦	www.vistaprint.ch - info@vistaprint.ch
¦___________________________________________________________________________________________________

Function desription:
Vacuum Pump implementation. 


History:
Version		Date			Author		Comment
---------------------------------------------------------------------------------------------------
0.00.1		09.07.2013		PC			Start history
0.00.2		19.02.2014		AVME/MRU	Changes in sta_TurnBusy for simulation
0.00.3		24.02.2014		AVME/MRU	sta_OFFBusy reworked

___________________________________________________________________________________________________*)

SUPER^();

(*
IF (me.bolActivate) THEN // cyclic call enabled
	IF (CIf.Info.bolInitDone=FALSE) THEN // first cycle -> init
		CtrlInit();
		CIf.Info.bolInitDone := TRUE;
	ELSE
		CycleStartDuty();
	
		Always();
		
		StateMachine();
		
		CycleEndDuty();
	END_IF
END_IF;
*)

PROPERTY ActualPosition : UINT
GET
ActualPosition := SIf.Cur.uintActualPosition;
END_GET
END_PROPERTY

METHOD PROTECTED Always : BOOL
SUPER^.Always();

// ----------------------------------------------------------------------------------
// cyclic actions outside of statemachine
IF (me.StateMachine.intState<>cSTA_SINGLE_ANSWER) THEN
	
	; // always error supervision
	
END_IF

// ----------------------------------------------------------------------------------
// Conditions Always
IF (((me.Alarm.eActivAlmClass=E_AlmClass.EOFF) OR (me.Alarm.eActivAlmClass=E_AlmClass.OFF) OR (me.intCmd=cCMD_OFF))
		 AND (me.StateMachine.intState<>cSTA_ERROR) AND (me.StateMachine.intState<>cSTA_ERRORQuit) AND
		(me.StateMachine.intState<>cSTA_OFF) AND (me.StateMachine.intState<>cSTA_OFFBusy)) THEN
	// alarm evt EOFF, OFF or cmd off
	me.StateMachine.intStateNext := cSTA_OFFBusy;
END_IF
END_METHOD

METHOD PUBLIC CtrlInit : BOOL
VAR_INPUT
END_VAR
SUPER^.CtrlInit();

// get child if
pMotor_CIF := AddChild(p_fbMotor^);
END_METHOD

PROPERTY PUBLIC CtrlSIf : POINTER TO T_Ctrl_SIf_MDC
GET
CtrlSIf := ADR(SIf);
END_GET
END_PROPERTY

PROPERTY PUBLIC Drive :  POINTER TO FB_UMC
GET
Drive := p_fbMotor;
END_GET
SET
p_fbMotor := Drive;
END_SET
END_PROPERTY

METHOD FB_init : BOOL
VAR_INPUT
	bInitRetains : BOOL; // if TRUE, the retain variables are initialized (warm start / cold start)
	bInCopyCode : BOOL;  // if TRUE, the instance afterwards gets moved into the copy code (online change)
END_VAR
VAR
	iIdx		: UINT;
	iLength		: UINT;	
END_VAR
//------------------------------------------------------------------------------------------------------------------------
// to manually change in new FUB implementation!!!
// define valid commands for this controller
iLength := SIZEOF(CIf.Job.aCmdList)/SIZEOF(CIf.Job.aCmdList[0]);
iIdx := 0;

WHILE (iIdx < iLength) AND (CIf.Job.aCmdList[iIdx].intCmd <> cCMD_INITIALIZED) DO
	iIdx := iIdx + 1; 
END_WHILE

IF (iIdx < iLength) THEN
// Add configuration of own comands	
	CIf.Job.aCmdList[iIdx].intCmd := MDC_CmdState.cCMD_INITIALIZE;
	CIf.Job.aCmdList[iIdx].strName := 'Initialize'; 
	CIf.Job.aCmdList[iIdx].bolAvailable := TRUE;
	iIdx := iIdx + 1;
	CIf.Job.aCmdList[iIdx].intCmd := MDC_CmdState.cCMD_TURN;
	CIf.Job.aCmdList[iIdx].strName := 'Turn'; 
	CIf.Job.aCmdList[iIdx].bolAvailable := TRUE;
	iIdx := iIdx + 1;
	CIf.Job.aCmdList[iIdx].intCmd := BASE_PLC.cCMD_RUN;
	CIf.Job.aCmdList[iIdx].strName := 'Run'; 
	CIf.Job.aCmdList[iIdx].bolAvailable := TRUE;
	iIdx := iIdx + 1;
	CIf.Job.aCmdList[iIdx].intCmd := MDC_CmdState.cCMD_PREPOSITION;
	CIf.Job.aCmdList[iIdx].strName := 'PrePosition'; 
	CIf.Job.aCmdList[iIdx].bolAvailable := TRUE;
	iIdx := iIdx + 1;
ELSE
	// Error if the aCmdList Array is to small
END_IF

// set name of class/typ
CIf.Info.strType := 'FB_MDC';
CIf.Info.strFullName := 'Malteser Drive Controller';

// set alarm class
SIf.Alm[E_ALM_MDC.TableSensorTimeout].eAlmClass := Base_PLC.E_AlmClass.TSTOP;
SIf.Alm[E_ALM_MDC.TableSensorTimeout].strText := 'Table Sensor Timeout'; 
SIf.Alm[E_ALM_MDC.CrossSensorTimeout].eAlmClass := Base_PLC.E_AlmClass.TSTOP;
SIf.Alm[E_ALM_MDC.CrossSensorTimeout].strText := 'Cross Sensor Timeout';
SIf.Alm[E_ALM_MDC.PositionSame].eAlmClass := Base_PLC.E_AlmClass.WARNING;
SIf.Alm[E_ALM_MDC.PositionSame].strText := 'New Position is the same as the actual position';

//*******************************************************************************
// initial values
//*******************************************************************************

// software configuration
CIf.SwCfg.bolExist := TRUE;
CIf.SwCfg.bolEnable := TRUE;
CIf.SwCfg.bolSimulation := FALSE;

// parameter
SIf.Cfg.uintPositionPerTurn			:= 4;
SIf.Par.intTurnDirection			:= 0;
SIf.Par.uinPositionToGo				:= 0;
SIf.Par.uinPositionSpeed_rpm		:= 1400;
SIf.Par.uinPrePositionSpeed_rpm		:= 450;
SIf.Par.udiInitializationTime_ms 	:= 16000;
SIf.Par.udiStepRotationTime_ms 		:= 2000;
SIf.Par.udiSimInitializationTime_ms := SIf.Par.udiInitializationTime_ms / 2;
SIf.Par.udiSimStepRotationTime_ms := SIf.Par.udiStepRotationTime_ms / 2;
SIf.Par.udiSimStartRotationTime_ms := SIf.Par.udiStepRotationTime_ms / 10;
END_METHOD

METHOD PROTECTED getCmdState : STRING

VAR_INPUT
	intCmdState: INT;
	bolState: BOOL;
END_VAR
getCmdState := SUPER^.getCmdState(intCmdState:=intCmdState,bolState:=bolState); // get global/base defined cmds/states

IF (getCmdState='') THEN // global not defined get local
	// get string cmd/state string information in runtime
	IF (bolState=FALSE) THEN
		CASE intCmdState OF
			MDC_CmdState.cCMD_INITIALIZE: 
				getCmdState := 'Initialize';
			MDC_CmdState.cCMD_TURN: 
				getCmdState := 'Turn';
			MDC_CmdState.cCMD_PREPOSITION: 
				getCmdState := 'PrePosition';
		END_CASE;
	ELSE
		// States's
		CASE intCmdState OF
			MDC_CmdState.cSTA_InitializeBusy: 
				getCmdState := 'InitializeBusy';
			MDC_CmdState.cSTA_InPositionBusy: 
				getCmdState := 'InPositionBusy';
			MDC_CmdState.cSTA_InPosition: 
				getCmdState := 'InPosition';
			MDC_CmdState.cSTA_StartTurnBusy: 
				getCmdState := 'StartTurnBusy';
			MDC_CmdState.cSTA_TurnBusy: 
				getCmdState := 'TurnBusy';
			MDC_CmdState.cSTA_TURNDONE: 
				getCmdState := 'TURNDONE';
			MDC_CmdState.cSTA_PREPOSITIONbusy: 
				getCmdState := 'PREPOSITIONbusy';
			MDC_CmdState.cSTA_PREPOSITION: 
				getCmdState := 'PREPOSITION';

			MDC_CmdState.cSUB_STOPbusy: 
				getCmdState := 'STOPbusy';
			MDC_CmdState.cSUB_TURNbusy: 
				getCmdState := 'TURNbusy';
			MDC_CmdState.cSUB_FINDHOLEbusy: 
				getCmdState := 'FINDHOLEbusy';
		END_CASE;
	END_IF
END_IF
END_METHOD

METHOD getCtrlSIf : POINTER TO T_Ctrl_SIf_MDC
getCtrlSIf := ADR(SIf);
END_METHOD

METHOD PROTECTED GetTurningDirection : E_TURN_DIRECTION
VAR
	iDifference 		: INT;
END_VAR
GetTurningDirection := E_TURN_DIRECTION.RIGHT;

// Determine the turning direction depending on set value or on shortest distance
CASE SIf.Par.intTurnDirection OF
	E_TURN_DIRECTION.LEFT	:
		GetTurningDirection := E_TURN_DIRECTION.LEFT;
	E_TURN_DIRECTION.AUTOMATIC 	:
		GetTurningDirection := E_TURN_DIRECTION.RIGHT;
		
		IF (SIf.Cur.uintActualPosition = 1) AND (SIf.Par.uinPositionToGo = 0) THEN
			iDifference := 0;
		END_IF

		iDifference := UINT_TO_INT(SIf.Par.uinPositionToGo - SIf.Cur.uintActualPosition);
		iDifference := ABS(iDifference);
		
		IF (    (SIf.Par.uinPositionToGo < SIf.Cur.uintActualPosition) AND (iDifference < UINT_TO_INT(SIf.Cfg.uintPositionPerTurn / 2)) 
			 OR (SIf.Par.uinPositionToGo > SIf.Cur.uintActualPosition) AND (iDifference > UINT_TO_INT(SIf.Cfg.uintPositionPerTurn / 2))) THEN
			GetTurningDirection := E_TURN_DIRECTION.LEFT;
		END_IF;
	E_TURN_DIRECTION.RIGHT	:
		GetTurningDirection := E_TURN_DIRECTION.RIGHT;
END_CASE;
END_METHOD

METHOD PROTECTED IncrementPosition : UINT
VAR_INPUT
	uinPosition		: UINT;
	eDirection		: E_TURN_DIRECTION;
END_VAR
VAR
	iNewPosition	: INT;
END_VAR
IF eDirection = E_TURN_DIRECTION.RIGHT THEN
	iNewPosition := UINT_TO_INT((uinPosition + 1) MOD SIf.Cfg.uintPositionPerTurn);
ELSE
	iNewPosition := UINT_TO_INT(uinPosition) - 1;
	
	IF (iNewPosition < 0) THEN
		iNewPosition := UINT_TO_INT(SIf.Cfg.uintPositionPerTurn) - 1;
	END_IF
END_IF

IncrementPosition := INT_TO_UINT(iNewPosition);
END_METHOD

METHOD PROTECTED IoInBridge : BOOL
// digitale and analoge inputs read from hardware or forcing
SIf.In.bolCrossPositionSensor.map := NOT THIS^.In_bolCrossPositionSensor;
SIf.In.bolTablePositionSensor.map := THIS^.In_bolTablePositionSensor;

IF (CIf.SwCfg.bolSimulation = FALSE) THEN
	getInBol(CIf.Job.bolIoForce,ADR(SIf.In.bolCrossPositionSensor));
	getInBol(CIf.Job.bolIoForce,ADR(SIf.In.bolTablePositionSensor));
ELSE
	//simulation of global IO
END_IF
END_METHOD

METHOD PROTECTED IoOutBridge : BOOL
VAR
	bolSwitchValvesOff: BOOL;
END_VAR
// digitale and analoge inputs read from hardware or forcing
IF (CIf.SwCfg.bolSimulation = FALSE) THEN
	setOutBol(CIf.Job.bolIoForce ,ADR(SIf.Out.intActualPosition));

	THIS^.Out_intActualPosition := SIf.Out.intActualPosition.map;
END_IF
END_METHOD

METHOD SetPositionToGo : BOOL
VAR_INPUT
	uinPositionToGo: UINT;
END_VAR
SIf.Par.uinPositionToGo := uinPositionToGo;

SetPositionToGo := uinPositionToGo = SIf.Cur.uintActualPosition;
END_METHOD

METHOD PROTECTED sta_ERROR : BOOL
// state implemetation
//--------------------------------------------------------------------------------------
// Entry action
	IF (me.StateMachine.intState<>me.StateMachine.intStateLastCycle) THEN
		me.StateMachine.intStateHistory := me.StateMachine.intStateLastCycle; // -> possibillity to go back to state before error
		me.StateMachine.intStateLastCycle := me.StateMachine.intState;
		pMotor_CIF^.Job.intACmd := BASE_PLC.cCMD_OFF;		
	END_IF


//--------------------------------------------------------------------------------------
// Cyclic action
	IF (me.StateMachine.intState=me.StateMachine.intStateLastCycle) THEN
		
		;
		
		
		// State Change Condition
		IF (CIf.Job.bolAlmReset = TRUE) THEN
			me.StateMachine.intStateNext := cSTA_ERRORQuit;
		END_IF
	END_IF




//--------------------------------------------------------------------------------------
// Exit action
	IF (me.StateMachine.intState<>me.StateMachine.intStateNext) THEN
		;
	END_IF
END_METHOD

METHOD PROTECTED sta_ERRORQuit : BOOL
// state implemetation
//--------------------------------------------------------------------------------------
// Entry action
	IF (me.StateMachine.intState<>me.StateMachine.intStateLastCycle) THEN
		me.StateMachine.intStateLastCycle := me.StateMachine.intState;
		
	END_IF


//--------------------------------------------------------------------------------------
// Cyclic action
	IF (me.StateMachine.intState=me.StateMachine.intStateLastCycle) THEN
		
		;
		// evtl. wait time if reset of device is necessary and then decide to go to states or ERROR state
		IF (CIf.Job.bolAlmReset = TRUE) THEN
			CIf.Job.eMe_ActivAlmClass := E_AlmClass.NONE; // reset feedback channel for parent
			CIf.Job.bolAlmReset := FALSE;
		END_IF
		
		// State Change Condition
		IF (CIf.Job.bolAlmReset = FALSE) THEN
			IF (me.StateMachine.intStateHistory<=cSTA_PON) THEN
				me.StateMachine.intStateNext := cSTA_PONBusy;
			ELSIF(me.intCmd=cCMD_OFF) THEN
				me.StateMachine.intStateNext := cSTA_OFFBusy;
			ELSIF(me.intCmd=cCMD_STOP) THEN
				me.StateMachine.intStateNext := cSTA_STOPBusy;
			ELSIF(me.intCmd=MDC_CmdState.cCMD_INITIALIZE) THEN
				me.StateMachine.intStateNext := MDC_CmdState.cSTA_InitializeBusy;
			ELSIF(me.intCmd=MDC_CmdState.cCMD_TURN) THEN
				me.StateMachine.intStateNext := MDC_CmdState.cSTA_InitializeBusy;
			END_IF
		END_IF
	END_IF




//--------------------------------------------------------------------------------------
// Exit action
	IF (me.StateMachine.intState<>me.StateMachine.intStateNext) THEN
		;
	END_IF
END_METHOD

METHOD PROTECTED sta_InitializeBusy : BOOL
VAR
	bCrossSensorPassed		: BOOL;
	bTableSensorPassed		: BOOL;
END_VAR
// state implemetation
//--------------------------------------------------------------------------------------
// Entry action
	IF (me.StateMachine.intState<>me.StateMachine.intStateLastCycle) THEN
		me.StateMachine.intStateLastCycle := me.StateMachine.intState;
		// Set Speed
		p_fbMotor^.CtrlSIf^.Par.uinSpeed_rpm := SIf.Par.uinPositionSpeed_rpm;
		pMotor_CIF^.Job.intACmd := UMC_CmdState.cCMD_RIGHT;		
		SIf.Cur.eActualTurningDirection := E_TURN_DIRECTION.RIGHT;

		fbSimulationTimer.IN := FALSE;
		fbSimulationTimer.PT := UDINT_TO_TIME(SIf.Par.udiSimInitializationTime_ms);
		fbSimulationTimer(); // set time/reset timer
		fbSimulationTimer.IN := TRUE; // start timer
		
		bCrossSensorPassed := FALSE;
		bTableSensorPassed := FALSE;
	END_IF


//--------------------------------------------------------------------------------------
// Cyclic action
	IF (me.StateMachine.intState=me.StateMachine.intStateLastCycle) THEN
		IF (CIf.SwCfg.bolSimulation) THEN
			fbSimulationTimer(); // simulation time

			IF (fbSimulationTimer.Q) THEN
				SIf.In.bolCrossPositionSensor.intern := TRUE;
				SIf.In.bolTablePositionSensor.intern := TRUE;				
			END_IF
		END_IF
		
		bCrossSensorPassed := bCrossSensorPassed OR SIf.In.bolCrossPositionSensor.intern;
		bTableSensorPassed := bTableSensorPassed OR SIf.In.bolTablePositionSensor.intern;
	
		IF (me.StateMachine.udiTimeInState_ms > SIf.Par.udiInitializationTime_ms) THEN
			IF NOT bCrossSensorPassed THEN
				pfbAlarmCtrl^.setAlarm(CIf.Info.intCtrlId,INT_TO_UINT(E_ALM_MDC.CrossSensorTimeout),0,ADR(SIf.Alm),E_AlmState.RST,CIf.Job.eMe_ActivAlmClass);
			END_IF
			
			IF NOT bTableSensorPassed THEN
				pfbAlarmCtrl^.setAlarm(CIf.Info.intCtrlId,INT_TO_UINT(E_ALM_MDC.TableSensorTimeout),0,ADR(SIf.Alm),E_AlmState.RST,CIf.Job.eMe_ActivAlmClass);
			END_IF
			
			me.StateMachine.intStateNext := Base_PLC.cSTA_ERROR;	
		END_IF

		IF SIf.In.bolCrossPositionSensor.intern AND SIf.In.bolTablePositionSensor.intern THEN
			me.StateMachine.intStateNext := MDC_CmdState.cSTA_InPositionBusy;
		END_IF
	END_IF


//--------------------------------------------------------------------------------------
// Exit action
	IF (me.StateMachine.intState<>me.StateMachine.intStateNext) THEN
		p_fbMotor^.CtrlSIf^.Par.uinSpeed_rpm := SIf.Par.uinPositionSpeed_rpm;
		SIf.Cur.uintActualPosition := 0;
	END_IF
END_METHOD

METHOD PROTECTED sta_InPosition : Bool
// state implemetation
//--------------------------------------------------------------------------------------
// Entry action
	IF (me.StateMachine.intState<>me.StateMachine.intStateLastCycle) THEN
		me.StateMachine.intStateLastCycle := me.StateMachine.intState;
		
		IF CIf.Job.intACmd = BASE_PLC.cCMD_RUN THEN
			CIf.Job.intACmd := cCMD_DONE;
		END_IF

		IF CIf.Job.intMCmd = BASE_PLC.cCMD_RUN THEN
			CIf.Job.intMCmd := cCMD_DONE;
		END_IF
	END_IF


//--------------------------------------------------------------------------------------
// Cyclic action
	IF (me.StateMachine.intState = me.StateMachine.intStateLastCycle) THEN
		CASE me.intCmd OF
			MDC_CmdState.cCMD_TURN,
			MDC_CmdState.cCMD_PREPOSITION:
//				IF SIf.Par.uinPositionToGo <> SIf.Cur.uintActualPosition THEN
//					SIf.Cur.eActualTurningDirection := GetTurningDirection();

					CASE me.intCmd OF
						MDC_CmdState.cCMD_TURN:
							me.StateMachine.intStateNext := MDC_CmdState.cSTA_StartTurnBusy;
						MDC_CmdState.cCMD_PREPOSITION:
							me.StateMachine.intStateNext := MDC_CmdState.cSTA_PREPOSITIONbusy;
					END_CASE
//				ELSE
//					CIf.Job.intACmd := cCMD_DONE;
//					CIf.Job.intMCmd := cCMD_DONE;
//					pfbAlarmCtrl^.setAlarm(CIf.Info.intCtrlId,INT_TO_UINT(E_ALM_MDC.PositionSame),0,ADR(SIf.Alm),E_AlmState.RST,CIf.Job.eMe_ActivAlmClass);
//				END_IF
				
			MDC_CmdState.cCMD_INITIALIZE:	
				me.StateMachine.intStateNext := MDC_CmdState.cSTA_InitializeBusy;
		END_CASE
	END_IF


//--------------------------------------------------------------------------------------
// Exit action
	IF (me.StateMachine.intState<>me.StateMachine.intStateNext) THEN
		;
	END_IF
END_METHOD

METHOD PROTECTED sta_InPositionBusy : BOOL
VAR_INPUT
END_VAR
// state implemetation
//--------------------------------------------------------------------------------------
// Entry action
	IF (me.StateMachine.intState<>me.StateMachine.intStateLastCycle) THEN
		me.StateMachine.intStateLastCycle := me.StateMachine.intState;
		pMotor_CIF^.Job.intACmd := BASE_PLC.cCMD_STOP;		
	END_IF


//--------------------------------------------------------------------------------------
// Cyclic action
	IF (me.StateMachine.intState=me.StateMachine.intStateLastCycle) THEN
		IF pMotor_CIF^.Job.intState = BASE_PLC.cSTA_STOP THEN
			me.StateMachine.intStateNext := MDC_CmdState.cSTA_InPosition;
		END_IF
	END_IF


//--------------------------------------------------------------------------------------
// Exit action
	IF (me.StateMachine.intState<>me.StateMachine.intStateNext) THEN
		;
	END_IF
END_METHOD

METHOD PROTECTED sta_OFF : BOOL
VAR_INPUT
END_VAR
// state implemetation
//--------------------------------------------------------------------------------------
// Entry action
	IF (me.StateMachine.intState<>me.StateMachine.intStateLastCycle) THEN
		me.StateMachine.intStateLastCycle := me.StateMachine.intState;

	END_IF


//--------------------------------------------------------------------------------------
// Cyclic action
	IF (me.StateMachine.intState=me.StateMachine.intStateLastCycle) THEN
		IF me.intCmd = MDC_CmdState.cCMD_INITIALIZE THEN
			me.StateMachine.intStateNext := MDC_CmdState.cSTA_InitializeBusy;
		END_IF
	END_IF


//--------------------------------------------------------------------------------------
// Exit action
	IF (me.StateMachine.intState<>me.StateMachine.intStateNext) THEN
		;
	END_IF
END_METHOD

METHOD PROTECTED sta_OFFBusy : BOOL
VAR_INPUT
END_VAR
// state implemetation
//--------------------------------------------------------------------------------------
// Entry action
	IF (me.StateMachine.intState<>me.StateMachine.intStateLastCycle) THEN
		me.StateMachine.intStateLastCycle := me.StateMachine.intState;
		pMotor_CIF^.Job.intACmd := BASE_PLC.cCMD_OFF;		
	END_IF


//--------------------------------------------------------------------------------------
// Cyclic action
	IF (me.StateMachine.intState=me.StateMachine.intStateLastCycle) THEN
		// Set commandos not only in entry action because of possible errors or manual/auto changes
		pMotor_CIF^.Job.intACmd := BASE_PLC.cCMD_OFF;		

		IF pMotor_CIF^.Job.intState = BASE_PLC.cSTA_OFF THEN
			me.StateMachine.intStateNext := BASE_PLC.cSTA_OFF;
		END_IF
	END_IF


//--------------------------------------------------------------------------------------
// Exit action
	IF (me.StateMachine.intState<>me.StateMachine.intStateNext) THEN
		;
	END_IF
END_METHOD

METHOD PROTECTED sta_PON : BOOL
VAR_INPUT
END_VAR
// state implemetation
//--------------------------------------------------------------------------------------
// Entry action
	IF (me.StateMachine.intState<>me.StateMachine.intStateLastCycle) THEN
		me.StateMachine.intStateLastCycle := me.StateMachine.intState;
		
	END_IF


//--------------------------------------------------------------------------------------
// Cyclic action
	IF (me.StateMachine.intState=me.StateMachine.intStateLastCycle) THEN
		;
	END_IF




//--------------------------------------------------------------------------------------
// Exit action
	IF (me.StateMachine.intState<>me.StateMachine.intStateNext) THEN
		;
	END_IF
END_METHOD

METHOD PROTECTED sta_PREPOSITION : BOOL
VAR_INPUT
END_VAR
// state implemetation
//--------------------------------------------------------------------------------------
// Entry action
IF (me.StateMachine.intState<>me.StateMachine.intStateLastCycle) THEN
	me.StateMachine.intStateLastCycle := me.StateMachine.intState;

	CIf.Job.intACmd := cCMD_DONE;
	CIf.Job.intMCmd := cCMD_DONE;
END_IF


//--------------------------------------------------------------------------------------
// Cyclic action
IF (me.StateMachine.intState=me.StateMachine.intStateLastCycle) THEN
	CASE me.intCmd OF
		MDC_CmdState.cCMD_INITIALIZE:
			me.StateMachine.intStateNext := MDC_CmdState.cSTA_InitializeBusy;
		MDC_CmdState.cCMD_TURN:
			me.StateMachine.intStateNext := MDC_CmdState.cSTA_StartTurnBusy;
		BASE_PLC.cCMD_RUN:
			me.StateMachine.intStateNext := MDC_CmdState.cSTA_InPositionBusy;
	END_CASE
END_IF


//--------------------------------------------------------------------------------------
// Exit action
IF (me.StateMachine.intState<>me.StateMachine.intStateNext) THEN
	;
END_IF
END_METHOD

METHOD PROTECTED sta_PREPOSITIONbusy : BOOL
VAR_INPUT
END_VAR
VAR
	eOldDirection		: BASE_ELEMENTS.E_TURN_DIRECTION;
END_VAR
// state implemetation
//--------------------------------------------------------------------------------------
// Entry action
IF (me.StateMachine.intState<>me.StateMachine.intStateLastCycle) THEN
	me.StateMachine.intStateLastCycle := me.StateMachine.intState;
	
	IF SIf.Par.uinPositionToGo <> SIf.Cur.uintActualPosition THEN
		eOldDirection := SIf.Cur.eActualTurningDirection;
		SIf.Cur.eActualTurningDirection := GetTurningDirection();

		// Set Speed
		p_fbMotor^.CtrlSIf^.Par.uinSpeed_rpm := SIf.Par.uinPrePositionSpeed_rpm;
		
		// Send the comand
		CASE SIf.Cur.eActualTurningDirection OF
			E_TURN_DIRECTION.LEFT:
				pMotor_CIF^.Job.intACmd := cCMD_LEFT;		
			E_TURN_DIRECTION.RIGHT:
				pMotor_CIF^.Job.intACmd := cCMD_RIGHT;		
		END_CASE

		fbSimulationTimer.IN := FALSE;
		fbSimulationTimer.PT := UDINT_TO_TIME(SIf.Par.udiSimStartRotationTime_ms);
		fbSimulationTimer(); // set time/reset timer
		fbSimulationTimer.IN := TRUE; // start timer
		
		IF eOldDirection = SIf.Cur.eActualTurningDirection THEN
			me.SubStateMachine.intState	    := MDC_CmdState.cSUB_TURNbusy;
			me.SubStateMachine.intStateNext := MDC_CmdState.cSUB_TURNbusy;
		ELSE
			me.SubStateMachine.intState	    := MDC_CmdState.cSUB_FINDHOLEbusy;
			me.SubStateMachine.intStateNext := MDC_CmdState.cSUB_FINDHOLEbusy;
		END_IF
	ELSE
		me.StateMachine.intStateNext := MDC_CmdState.cSTA_PREPOSITION;
	END_IF
END_IF


//--------------------------------------------------------------------------------------
// Cyclic action
IF (me.StateMachine.intState=me.StateMachine.intStateLastCycle) THEN
	IF (CIf.SwCfg.bolSimulation) THEN
		fbSimulationTimer(); // simulation time

		IF (fbSimulationTimer.Q) THEN
			SIf.In.bolCrossPositionSensor.intern := FALSE;
			SIf.In.bolTablePositionSensor.intern := FALSE;
		END_IF
	END_IF
	
	CASE me.SubStateMachine.intState OF
		MDC_CmdState.cSUB_FINDHOLEbusy:
			IF SIf.In.bolCrossPositionSensor.intern THEN
				me.SubStateMachine.intStateNext := MDC_CmdState.cSUB_TURNbusy;
			END_IF
		MDC_CmdState.cSUB_TURNbusy:
			IF NOT SIf.In.bolCrossPositionSensor.intern THEN
				pMotor_CIF^.Job.intACmd := BASE_PLC.cCMD_STOP;		
				me.SubStateMachine.intStateNext := MDC_CmdState.cSUB_STOPbusy;
			END_IF
		MDC_CmdState.cSUB_STOPbusy:
			IF pMotor_CIF^.Job.intState = BASE_PLC.cSTA_STOP THEN
				me.StateMachine.intStateNext := MDC_CmdState.cSTA_PREPOSITION;
			END_IF
	END_CASE
	
	IF me.intCmd = MDC_CmdState.cCMD_TURN THEN
		IF SIf.Par.uinPositionToGo <> SIf.Cur.uintActualPosition THEN
			me.StateMachine.intStateNext := MDC_CmdState.cSTA_StartTurnBusy;
		ELSE
			CIf.Job.intACmd := cCMD_DONE;
			CIf.Job.intMCmd := cCMD_DONE;
			pfbAlarmCtrl^.setAlarm(CIf.Info.intCtrlId,INT_TO_UINT(E_ALM_MDC.PositionSame),0,ADR(SIf.Alm),E_AlmState.RST,CIf.Job.eMe_ActivAlmClass);
		END_IF
	END_IF

	IF (me.StateMachine.udiTimeInState_ms > SIf.Par.udiStepRotationTime_ms) THEN
		pfbAlarmCtrl^.setAlarm(CIf.Info.intCtrlId,INT_TO_UINT(E_ALM_MDC.CrossSensorTimeout),0,ADR(SIf.Alm),E_AlmState.RST,CIf.Job.eMe_ActivAlmClass);
		me.StateMachine.intStateNext := Base_PLC.cSTA_ERROR;	
	END_IF
	
	
END_IF


//--------------------------------------------------------------------------------------
// Exit action
IF (me.StateMachine.intState<>me.StateMachine.intStateNext) THEN
	;
END_IF
END_METHOD

METHOD PROTECTED sta_StartTurnBusy : Bool
VAR
	iDifference			: INT;
	eOldDirection		: BASE_ELEMENTS.E_TURN_DIRECTION;
END_VAR
// state implemetation
//--------------------------------------------------------------------------------------
// Entry action
	IF (me.StateMachine.intState<>me.StateMachine.intStateLastCycle) THEN
		me.StateMachine.intStateLastCycle := me.StateMachine.intState;
		
		IF SIf.Par.uinPositionToGo <> SIf.Cur.uintActualPosition THEN
			eOldDirection := SIf.Cur.eActualTurningDirection;
			SIf.Cur.eActualTurningDirection := GetTurningDirection();

			// Set Speed
			p_fbMotor^.CtrlSIf^.Par.uinSpeed_rpm := SIf.Par.uinPositionSpeed_rpm;
			
			// Send the comand
			CASE SIf.Cur.eActualTurningDirection OF
				E_TURN_DIRECTION.LEFT:
					pMotor_CIF^.Job.intACmd := cCMD_LEFT;		
				E_TURN_DIRECTION.RIGHT:
					pMotor_CIF^.Job.intACmd := cCMD_RIGHT;		
			END_CASE

			IF eOldDirection = SIf.Cur.eActualTurningDirection THEN
				me.SubStateMachine.intState	    := MDC_CmdState.cSUB_TURNbusy;
				me.SubStateMachine.intStateNext := MDC_CmdState.cSUB_TURNbusy;
			ELSE
				me.SubStateMachine.intState	    := MDC_CmdState.cSUB_FINDHOLEbusy;
				me.SubStateMachine.intStateNext := MDC_CmdState.cSUB_FINDHOLEbusy;
			END_IF
			
			fbSimulationTimer.IN := FALSE;
			fbSimulationTimer.PT := UDINT_TO_TIME(SIf.Par.udiSimStartRotationTime_ms);
			fbSimulationTimer(); // set time/reset timer
			fbSimulationTimer.IN := TRUE; // start timer
		END_IF
	END_IF


//--------------------------------------------------------------------------------------
// Cyclic action
	IF (me.StateMachine.intState=me.StateMachine.intStateLastCycle) THEN
		IF (CIf.SwCfg.bolSimulation) THEN
			fbSimulationTimer(); // simulation time

			IF (fbSimulationTimer.Q) THEN
				SIf.In.bolCrossPositionSensor.intern := FALSE;
				SIf.In.bolTablePositionSensor.intern := FALSE;
			END_IF
		END_IF
		
		CASE me.SubStateMachine.intState OF
			MDC_CmdState.cSUB_FINDHOLEbusy:
				IF SIf.In.bolCrossPositionSensor.intern THEN
					me.SubStateMachine.intStateNext := MDC_CmdState.cSUB_TURNbusy;
				END_IF
			MDC_CmdState.cSUB_TURNbusy:
				IF NOT SIf.In.bolCrossPositionSensor.intern THEN
					me.StateMachine.intStateNext := MDC_CmdState.cSTA_TurnBusy;
				END_IF
		END_CASE

		IF SIf.Par.uinPositionToGo = SIf.Cur.uintActualPosition THEN
			me.StateMachine.intStateNext := MDC_CmdState.cSTA_TURNDONE;
		END_IF 
		
		IF (me.StateMachine.udiTimeInState_ms > SIf.Par.udiStepRotationTime_ms) THEN
			pfbAlarmCtrl^.setAlarm(CIf.Info.intCtrlId,INT_TO_UINT(E_ALM_MDC.CrossSensorTimeout),0,ADR(SIf.Alm),E_AlmState.RST,CIf.Job.eMe_ActivAlmClass);
			me.StateMachine.intStateNext := Base_PLC.cSTA_ERROR;	
		END_IF
	END_IF


//--------------------------------------------------------------------------------------
// Exit action
	IF (me.StateMachine.intState<>me.StateMachine.intStateNext) THEN
		;
	END_IF
END_METHOD

METHOD PROTECTED sta_TurnBusy : Bool
VAR_INPUT
END_VAR
// state implemetation
//--------------------------------------------------------------------------------------
// Entry action
	IF (me.StateMachine.intState<>me.StateMachine.intStateLastCycle) THEN
		me.StateMachine.intStateLastCycle := me.StateMachine.intState;

		fbSimulationTimer.IN := FALSE;
		fbSimulationTimer.PT := UDINT_TO_TIME(SIf.Par.udiSimStepRotationTime_ms);
		fbSimulationTimer(); // set time/reset timer
		fbSimulationTimer.IN := TRUE; // start timer

		me.SubStateMachine.intState 	:= MDC_CmdState.cSUB_TURNbusy;
		me.SubStateMachine.intStateNext := MDC_CmdState.cSUB_TURNbusy;
	END_IF


//--------------------------------------------------------------------------------------
// Cyclic action
	IF (me.StateMachine.intState=me.StateMachine.intStateLastCycle) THEN
		IF (CIf.SwCfg.bolSimulation) THEN
			fbSimulationTimer(); // simulation time

			IF (fbSimulationTimer.Q) THEN
				SIf.In.bolCrossPositionSensor.intern := TRUE;
			END_IF
		END_IF
		
		CASE me.SubStateMachine.intState OF
			MDC_CmdState.cSUB_TURNbusy:
				IF SIf.In.bolCrossPositionSensor.intern THEN
					SIf.Cur.uintActualPosition := IncrementPosition(SIf.Cur.uintActualPosition,SIf.Cur.eActualTurningDirection);
					
					IF (CIf.SwCfg.bolSimulation) THEN
						IF SIf.Cur.uintActualPosition = 0 THEN
							SIf.In.bolTablePositionSensor.intern := TRUE;
						END_IF
					END_IF
					
					IF SIf.Par.uinPositionToGo = SIf.Cur.uintActualPosition THEN
						pMotor_CIF^.Job.intACmd := BASE_PLC.cCMD_STOP;		
						me.SubStateMachine.intStateNext := MDC_CmdState.cSUB_STOPbusy;
					ELSE
						me.StateMachine.intStateNext := MDC_CmdState.cSTA_StartTurnBusy;
					END_IF 
				END_IF
				
			MDC_CmdState.cSUB_STOPbusy:
				IF pMotor_CIF^.Job.intState = BASE_PLC.cSTA_STOP THEN
					me.StateMachine.intStateNext := MDC_CmdState.cSTA_TURNDONE;
				END_IF
		END_CASE


		IF (me.StateMachine.udiTimeInState_ms > SIf.Par.udiStepRotationTime_ms) THEN
			pfbAlarmCtrl^.setAlarm(CIf.Info.intCtrlId,INT_TO_UINT(E_ALM_MDC.CrossSensorTimeout),0,ADR(SIf.Alm),E_AlmState.RST,CIf.Job.eMe_ActivAlmClass);
			me.StateMachine.intStateNext := Base_PLC.cSTA_ERROR;	
		END_IF
	END_IF


//--------------------------------------------------------------------------------------
// Exit action
	IF (me.StateMachine.intState<>me.StateMachine.intStateNext) THEN
		;
	END_IF
END_METHOD

METHOD PROTECTED sta_TURNDONE : BOOL
VAR_INPUT
END_VAR
// state implemetation
//--------------------------------------------------------------------------------------
// Entry action
IF (me.StateMachine.intState<>me.StateMachine.intStateLastCycle) THEN
	me.StateMachine.intStateLastCycle := me.StateMachine.intState;
	
	IF CIf.Job.intACmd = MDC_CmdState.cCMD_TURN THEN
		CIf.Job.intACmd := cCMD_DONE;
	END_IF
	
	IF CIf.Job.intMCmd = MDC_CmdState.cCMD_TURN THEN
		CIf.Job.intMCmd := cCMD_DONE;
	END_IF
END_IF


//--------------------------------------------------------------------------------------
// Cyclic action
IF (me.StateMachine.intState=me.StateMachine.intStateLastCycle) THEN
	CASE me.intCmd OF
		MDC_CmdState.cCMD_INITIALIZE:
			me.StateMachine.intStateNext := MDC_CmdState.cSTA_InitializeBusy;
		BASE_PLC.cCMD_RUN:
			me.StateMachine.intStateNext := MDC_CmdState.cSTA_InPositionBusy;
	END_CASE
END_IF


//--------------------------------------------------------------------------------------
// Exit action
IF (me.StateMachine.intState<>me.StateMachine.intStateNext) THEN
	;
END_IF
END_METHOD

METHOD PROTECTED StateMachine : BOOL
SUPER^.StateMachine();

// main statemachine of base controller
CASE me.StateMachine.intState OF
    MDC_CmdState.cSTA_InitializeBusy: 
        THIS^.sta_InitializeBusy();
    MDC_CmdState.cSTA_InPositionBusy: 
        THIS^.sta_InPositionBusy();
    MDC_CmdState.cSTA_InPosition: 
        THIS^.sta_InPosition();
    MDC_CmdState.cSTA_StartTurnBusy: 
        THIS^.sta_StartTurnBusy();
    MDC_CmdState.cSTA_TurnBusy: 
        THIS^.sta_TurnBusy();
    MDC_CmdState.cSTA_PREPOSITION: 
        THIS^.sta_PREPOSITION();
    MDC_CmdState.cSTA_PREPOSITIONbusy: 
        THIS^.sta_PREPOSITIONbusy();
    MDC_CmdState.cSTA_TURNDONE: 
        THIS^.sta_TURNDONE();
END_CASE;
END_METHOD

END_FUNCTION_BLOCK

// POUs/Controller/Lvl1/OVN (Oven)/helper/cycle_Ovn
FUNCTION cycle_Ovn : BOOL
VAR_INPUT
	pOvn: POINTER TO T_OVN;
END_VAR

pOvn^.ctrl.fbOvn_Ibh();

pOvn^.ctrl.fbOvn.In_iStatus := pOvn^.ctrl.fbOvn_Ibh.Out_iStatus;
pOvn^.ctrl.fbOvn.In_bOff := pOvn^.ctrl.fbOvn_Ibh.Out_bOff;
pOvn^.ctrl.fbOvn.In_bBeltOn := pOvn^.ctrl.fbOvn_Ibh.Out_bBeltOn;
pOvn^.ctrl.fbOvn.In_bManual := pOvn^.ctrl.fbOvn_Ibh.Out_bManual;
pOvn^.ctrl.fbOvn.In_bRun := pOvn^.ctrl.fbOvn_Ibh.Out_bRun;
pOvn^.ctrl.fbOvn.In_bAckError := pOvn^.ctrl.fbOvn_Ibh.Out_bAckError;
pOvn^.ctrl.fbOvn.In_adiTemp_dc := pOvn^.ctrl.fbOvn_Ibh.Out_adiTemp_dc;
pOvn^.ctrl.fbOvn.In_adiAir_p := pOvn^.ctrl.fbOvn_Ibh.Out_adiAir_p;
pOvn^.ctrl.fbOvn.In_diSpeed_mm_min := pOvn^.ctrl.fbOvn_Ibh.Out_diSpeed_mm_min;
pOvn^.ctrl.fbOvn.In_iErrorLevel := pOvn^.ctrl.fbOvn_Ibh.Out_iErrorLevel;
pOvn^.ctrl.fbOvn.In_iErrorID := pOvn^.ctrl.fbOvn_Ibh.Out_iErrorID;
pOvn^.ctrl.fbOvn.In_bDriverConnected := pOvn^.ctrl.fbOvn_Ibh.Out_bDriverConnected;
pOvn^.ctrl.fbOvn.In_bDriverError := pOvn^.ctrl.fbOvn_Ibh.Out_bDriverError;
pOvn^.ctrl.fbOvn.In_udiDriverErrorID := pOvn^.ctrl.fbOvn_Ibh.Out_udiDriverErrorID;

//... := pOvn^.io.In_bolBcrDistributionTrigger;	//TODO
pOvn^.ctrl.fbOvn.In_uliBarcodeNew_1 := pOvn^.io.In_udiBarcode_new_1;
pOvn^.ctrl.fbOvn.In_uliBarcodeNew_2 := pOvn^.io.In_udiBarcode_new_2;
pOvn^.ctrl.fbOvn.In_uiNewElement_1 := pOvn^.io.In_uinNew_element_1;
pOvn^.ctrl.fbOvn.In_uiNewElement_2 := pOvn^.io.In_uinNew_element_2;
pOvn^.ctrl.fbOvn.In_uliBarcodeDelete_1 := pOvn^.io.In_udiBarcode_delete_1;
pOvn^.ctrl.fbOvn.In_uliBarcodeDelete_2 := pOvn^.io.In_udiBarcode_delete_2;
pOvn^.ctrl.fbOvn.In_uiDeleteElement_1 := pOvn^.io.In_uinDelete_element_1;
pOvn^.ctrl.fbOvn.In_uiDeleteElement_2 := pOvn^.io.In_uinDelete_element_2;

pOvn^.ctrl.fbOvn();

//pOvn^.io.Out_uinBcrOvenAEvent := ...;	//TODO
//pOvn^.io.Out_udiBcrOvenACode := ...;	//TODO
//pOvn^.io.Out_uinBcrOvenBEvent := ...;	//TODO
//pOvn^.io.Out_udiBcrOvenBCode := ...;	//TODO

pOvn^.datachn.rSendData.fbFifo();

END_FUNCTION

// POUs/Controller/Lvl1/OVN (Oven)/helper/init_Ovn
FUNCTION init_Ovn : BOOL
VAR_INPUT
	pOvn			: POINTER TO T_OVN;
	/// instance array of all controller instances
	pCtrlInst		: POINTER TO fb_CtrlBase;
	/// common interface array of all controllers (main use for PLC)
	pCtrlCIf		: POINTER TO T_Ctrl_CIf;
END_VAR

pOvn^.datachn.rSendData.fbDataChannel.InitChannel(SIZEOF(pOvn^.datachn.rSendData.rDataChannelItem), ADR(pOvn^.datachn.rSendData.rDataChannelItem));
pOvn^.datachn.rSendData.fbFifo.DataChannel := ADR(pOvn^.datachn.rSendData.fbDataChannel);
pOvn^.datachn.rSendData.fbFifo.FreeDataPointer := TRUE;
pOvn^.datachn.rSendData.fbFifo.Enable := TRUE;

pOvn^.ctrl.fbOvn_Ibh.iniAllCtrlArrays(pCtrlInst,pCtrlCIf,pOvn^.id.Ovn_Ibh);
pOvn^.ctrl.fbOvn.iniAllCtrlArrays(pCtrlInst,pCtrlCIf,pOvn^.id.Ovn);
pOvn^.ctrl.fbOvn.IBH := ADR(pOvn^.ctrl.fbOvn_Ibh);
pOvn^.ctrl.fbOvn.DataChannel := ADR(pOvn^.datachn.rSendData.fbFifo);

END_FUNCTION

// POUs/Controller/Lvl1/OVN (Oven)/FB_MONITOR
FUNCTION_BLOCK FB_MONITOR
VAR_INPUT
	diCurrentValue: DINT;
	diTargetValue: DINT;
	diBand1: DINT;
	diBand2: DINT;
	udiTimeout_ms: UDINT;
	udiSampleTime_ms: UDINT := 0;
END_VAR
VAR_OUTPUT
	bOutOfBand: BOOL;
	bError: BOOL;
END_VAR
VAR
	udiTimeOutOfBand_ms: UDINT := 0;
END_VAR

bError := FALSE;
bOutOfBand := FALSE;

// Band 1
IF (ABS(diCurrentValue - diTargetValue) > ABS(diBand1)) THEN
	bOutOfBand := TRUE;
	udiTimeOutOfBand_ms := udiTimeOutOfBand_ms + udiSampleTime_ms;
	IF (udiTimeOutOfBand_ms > udiTimeout_ms) THEN
		bError := TRUE;
	END_IF
ELSE
	udiTimeOutOfBand_ms := 0;
END_IF

// Band 2
IF (ABS(diCurrentValue - diTargetValue) > ABS(diBand2)) THEN
	bOutOfBand := TRUE;
	bError := TRUE;
END_IF

ACTION resetTime:
THIS^.udiTimeOutOfBand_ms := 0;
END_ACTION

END_FUNCTION_BLOCK

// POUs/Controller/Lvl1/OVN (Oven)/FB_OVN
FUNCTION_BLOCK FB_OVN EXTENDS FB_CtrlBase
VAR_INPUT
	/// 0 = Busy, 1 = OFF, 2 = BeltOn, 3 = Manual, 4 = Run, 5 = Error, 6 = Bundverschlusserkennung 
	In_iStatus: INT;
	/// Machine off 
	In_bOff: BOOL;
	/// Band on 
	In_bBeltOn: BOOL;
	/// Manual 
	In_bManual: BOOL;
	/// Standart drying process 
	In_bRun: BOOL;
	/// Resetting error 
	In_bAckError: BOOL;
	/// Actual temperature in deci °C 
	In_adiTemp_dc: ARRAY[0..(MAX_NUMBER_OF_OVEN_MODULES - 1)] OF DINT;
	/// Aactual airflow in % 
	In_adiAir_p: ARRAY[0..(MAX_NUMBER_OF_OVEN_MODULES - 1)] OF DINT;
	/// Actual belt speed in mm/min 
	In_diSpeed_mm_min: DINT;
	/// 1=Information, 2=Warning, 3=Error 
	In_iErrorLevel: INT;
	/// Error ID (e.g. 100=temperature overflow) 
	In_iErrorID: INT;
	In_bDriverConnected: BOOL;
	In_bDriverError: BOOL;
	In_udiDriverErrorID: UDINT;
	In_uliBarcodeNew_1: ULINT;
	In_uliBarcodeNew_2: ULINT;
	In_uiNewElement_1: UINT;
	In_uiNewElement_2: UINT;
	In_uliBarcodeDelete_1: ULINT;
	In_uliBarcodeDelete_2: ULINT;
	In_uiDeleteElement_1: UINT;
	In_uiDeleteElement_2: UINT;
END_VAR
VAR
	/// Specific interface struct for public access
	SIf: T_Ctrl_SIf_OVN;
	/// this allows to detect parameter changes
	lastSifPar: T_Ctrl_SIf_OVN_Par;
	/// pointer to function block
	p_fbIBH: POINTER TO FB_IBH;
	p_fbIBH_CIf: POINTER TO BASE_PLC.T_Ctrl_CIf;
	/// Monitors
	afbTempMonitors: ARRAY[0..(MAX_NUMBER_OF_OVEN_MODULES - 1)] OF FB_MONITOR;
	afbAirMonitors: ARRAY[0..(MAX_NUMBER_OF_OVEN_MODULES - 1)] OF FB_MONITOR;
	fbSpeedMonitor: FB_MONITOR;
	udiTimeInBand: UDINT;
	/// Tracker
	fbTracker: FB_Tracker;
	/// Error Tracking
	iLastCalledAlarmNr: INT;
	uiNewElementOld_1: UINT;
	uiNewElementOld_2: UINT;
	uiDeleteElementOld_1: UINT;
	uiDeleteElementOld_2: UINT;
	
	bSimLastCycle: BOOL;
END_VAR

(*__________________________________________________________________________________________________
¦	
¦	Vistaprint Schweiz GmbH
¦	CH - 8401 Winterthur
¦
¦	www.vistaprint.ch - info@vistaprint.ch
¦___________________________________________________________________________________________________

Function desription:
Oven Controller Implementation

History:
Version		Date			Author		Comment
---------------------------------------------------------------------------------------------------
0.00.1		10.12.2013		BB			Start history
___________________________________________________________________________________________________*)

// check if child pointer valid
IF (me.bolActivate) THEN // cyclic call enabled
	
	IF (CIf.Info.bolInitDone=FALSE) THEN // first cycle -> init
		CtrlInit();
		CIf.Info.bolInitDone := TRUE;
	ELSE
		CycleStartDuty();
		
		Always();
		
		StateMachine();
		
		CycleEndDuty();
	END_IF
	
END_IF;

{attribute 'object_name' := 'Always'}
METHOD PROTECTED Always : BOOL
VAR
	fbOVN: INT;
	bResettable: BOOL;
END_VAR
SUPER^.Always();

// ----------------------------------------------------------------------------------
// cyclic actions outside of statemachine
IF (me.StateMachine.intState<>cSTA_SINGLE_ANSWER) THEN
	
	// copy number of modules to IBH driver
	p_fbIBH^.getCtrlSIf()^.Cfg.uiNumberOfModules := SIf.Cfg.uiNumberOfModules;
	
	// Simulation
	IF (CIf.SwCfg.bolSimulation) THEN
		p_fbIBH^.CtrlCIf^.SwCfg.bolEnable := FALSE;
	ELSE
		p_fbIBH^.CtrlCIf^.SwCfg.bolEnable := TRUE;
		IF bSimLastCycle THEN
			me.StateMachine.intState := cSTA_PONBusy;
			me.StateMachine.intStateNext := cSTA_PONBusy;
		END_IF
	END_IF
	bSimLastCycle := CIf.SwCfg.bolSimulation;
	
	// check parameter from GUI
	THIS^.checkParameter();
	
	// write input values directly to SIf.Cur
	SIf.Cur.diSpeed_mm_min := THIS^.In_diSpeed_mm_min;
	SIf.Cur.adiAir_p := THIS^.In_adiAir_p;
	SIf.Cur.adiTemp_dc := THIS^.In_adiTemp_dc;
	
	// remove old elements from Tracker
	IF In_uiDeleteElement_1<>uiDeleteElementOld_1 THEN
		uiDeleteElementOld_1 := In_uiDeleteElement_1;
		fbTracker.deleteElement(In_uliBarcodeDelete_1, SIf.Cfg.bolDataChannelEnable);
	END_IF
	IF In_uiDeleteElement_2<>uiDeleteElementOld_2 THEN
		uiDeleteElementOld_2 := In_uiDeleteElement_2;
		fbTracker.deleteElement(In_uliBarcodeDelete_2, SIf.Cfg.bolDataChannelEnable);
	END_IF
	
	// update Tracker
	fbTracker.update(In_adiTemp_mc:=In_adiTemp_dc, In_diSpeed_mm_min:=In_diSpeed_mm_min,bolSendToSaber:=SIf.Cfg.bolDataChannelEnable);
	
	// add new elements to Tracker
	IF In_uiNewElement_1<>uiNewElementOld_1 THEN
		uiNewElementOld_1 := In_uiNewElement_1;
		fbTracker.addElement(In_uliBarcodeNew_1);
	END_IF
	IF In_uiNewElement_2<>uiNewElementOld_2 THEN
		uiNewElementOld_2 := In_uiNewElement_2;
		fbTracker.addElement(In_uliBarcodeNew_2);
	END_IF
	
	// check errors when higher than PONBusy
	IF (me.StateMachine.intState>=Base_PLC.cSTA_PON) AND (NOT CIf.SwCfg.bolSimulation) THEN
		
		// go to error if Driver connection is lost
		IF 		NOT THIS^.In_bDriverConnected
			AND	me.StateMachine.intState<>Base_PLC.cSTA_ERROR
			AND	me.StateMachine.intState<>Base_PLC.cSTA_ERRORQuit THEN
				pfbAlarmCtrl^.setAlarm(CIf.Info.intCtrlId,INT_TO_UDINT(E_ALM_OVN.ConnectionError),UDINT_TO_DINT(THIS^.In_udiDriverErrorID),ADR(SIf.Alm),E_AlmState.RST,CIf.Job.eMe_ActivAlmClass);
				me.StateMachine.intStateNext := Base_PLC.cSTA_ERROR;
				iLastCalledAlarmNr := E_ALM_OVN.ConnectionError;
		END_IF
		
		// check Tesoma Errors, ErrorLevel 1 (Info) and 2 (Warning) don't exist
		IF THIS^.In_iErrorLevel=3 THEN
			chooseTesomaErrors(bResettable);
			IF 		me.StateMachine.intState<>Base_PLC.cSTA_ERROR
				AND	me.StateMachine.intState<>Base_PLC.cSTA_ERRORQuit
				and me.StateMachine.intStateNext<>Base_PLC.cSTA_ERROR THEN
					me.StateMachine.intStateNext := Base_PLC.cSTA_ERROR;
			END_IF
		END_IF
		
	END_IF
	
END_IF

// ----------------------------------------------------------------------------------
// overrule error always from base -> no EOFF State!! in EOFF go to OFF
IF (me.StateMachine.intStateNext = cSTA_EOFFBusy) THEN
	IF (me.StateMachine.intState = cSTA_OFF) THEN
		me.StateMachine.intStateNext := cSTA_OFF;
	ELSE // stay in OFF
		me.StateMachine.intStateNext := cSTA_OFFBusy;
	END_IF
END_IF
END_METHOD

{attribute 'object_name' := 'checkParameter'}
METHOD checkParameter : BOOL
VAR
	uiIdx: UINT;
END_VAR
// Belt Speed
IF (SIf.Par.diSpeed_mm_min > SIf.Cfg.diMaxSpeed_mm_min) THEN
	pfbAlarmCtrl^.setAlarm(CIf.Info.intCtrlId,INT_TO_UDINT(E_ALM_OVN.ParameterWarning),0,ADR(SIf.Alm),E_AlmState.RST,CIf.Job.eMe_ActivAlmClass);
	SIf.Par.diSpeed_mm_min := SIf.Cfg.diMaxSpeed_mm_min;
ELSIF (SIf.Par.diSpeed_mm_min < SIf.Cfg.diMinSpeed_mm_min) THEN
	pfbAlarmCtrl^.setAlarm(CIf.Info.intCtrlId,INT_TO_UDINT(E_ALM_OVN.ParameterWarning),0,ADR(SIf.Alm),E_AlmState.RST,CIf.Job.eMe_ActivAlmClass);
	SIf.Par.diSpeed_mm_min := SIf.Cfg.diMinSpeed_mm_min;
END_IF

// Temperature
FOR uiIdx:=0 TO SIf.Cfg.uiNumberOfModules-1 BY 1 DO
	IF (SIf.Par.adiTemp_dc[uiIdx] > SIf.Cfg.diMaxTemp_dc) THEN
		pfbAlarmCtrl^.setAlarm(CIf.Info.intCtrlId,INT_TO_UDINT(E_ALM_OVN.ParameterWarning),uiIdx,ADR(SIf.Alm),E_AlmState.RST,CIf.Job.eMe_ActivAlmClass);
		SIf.Par.adiTemp_dc[uiIdx] := SIf.Cfg.diMaxTemp_dc;
	ELSIF (SIf.Par.adiTemp_dc[uiIdx] < SIf.Cfg.diMinTemp_dc) THEN
		pfbAlarmCtrl^.setAlarm(CIf.Info.intCtrlId,INT_TO_UDINT(E_ALM_OVN.ParameterWarning),uiIdx,ADR(SIf.Alm),E_AlmState.RST,CIf.Job.eMe_ActivAlmClass);
		SIf.Par.adiTemp_dc[uiIdx] := SIf.Cfg.diMinTemp_dc;
	END_IF
END_FOR

// Airflow
FOR uiIdx:=0 TO SIf.Cfg.uiNumberOfModules-1 BY 1 DO
	IF (SIf.Par.adiAir_p[uiIdx] > SIf.Cfg.diMaxAir_p) THEN
		pfbAlarmCtrl^.setAlarm(CIf.Info.intCtrlId,INT_TO_UDINT(E_ALM_OVN.ParameterWarning),uiIdx,ADR(SIf.Alm),E_AlmState.RST,CIf.Job.eMe_ActivAlmClass);
		SIf.Par.adiAir_p[uiIdx] := SIf.Cfg.diMaxAir_p;
	ELSIF (SIf.Par.adiAir_p[uiIdx] < SIf.Cfg.diMinAir_p) THEN
		pfbAlarmCtrl^.setAlarm(CIf.Info.intCtrlId,INT_TO_UDINT(E_ALM_OVN.ParameterWarning),uiIdx,ADR(SIf.Alm),E_AlmState.RST,CIf.Job.eMe_ActivAlmClass);
		SIf.Par.adiAir_p[uiIdx] := SIf.Cfg.diMinAir_p;
	END_IF
END_FOR
END_METHOD

{attribute 'object_name' := 'chooseTesomaErrors'}
METHOD chooseTesomaErrors : BOOL
VAR_IN_OUT
	bResettable: BOOL;
END_VAR
bResettable := FALSE;

